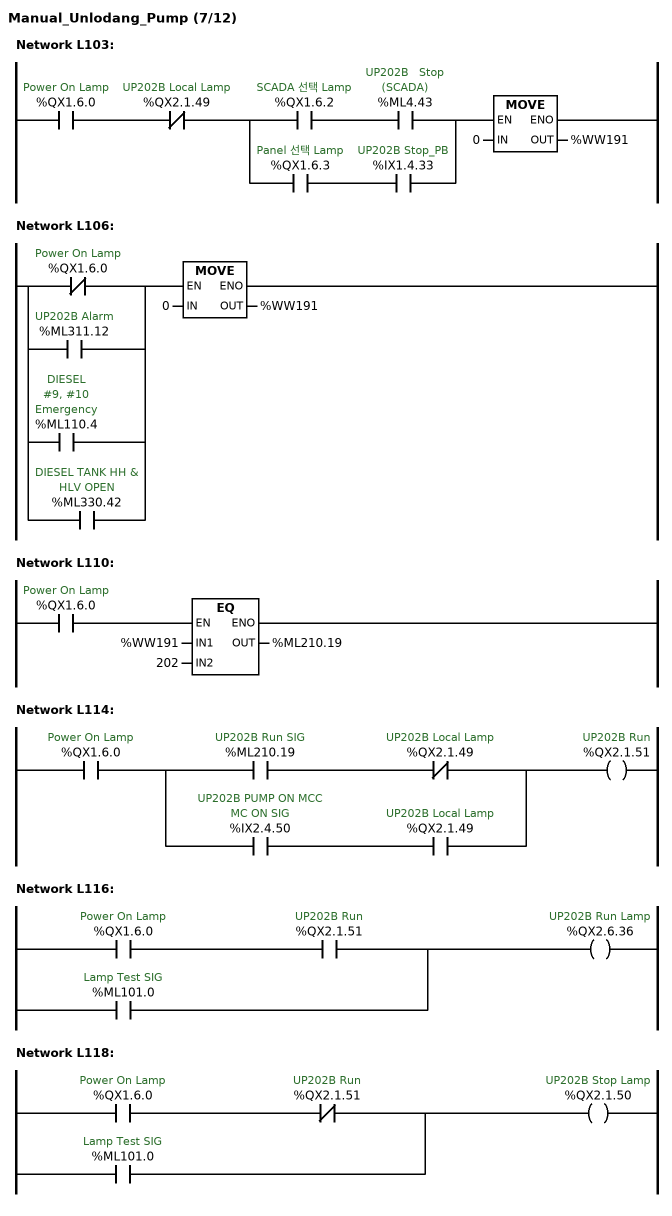
(* [picture p96: Manual_Unlodang_Pump rungs L103-L118] *)
(* Rung L103 *)
IF %QX1.6.0 AND NOT %QX2.1.49 AND ((%QX1.6.2 AND %ML4.43) OR (%QX1.6.3 AND %IX1.4.33)) THEN
    %WW191 := 0;
END_IF;
(* Rung L106 *)
IF NOT %QX1.6.0 OR %ML311.12 OR %ML110.4 OR %ML330.42 THEN %WW191 := 0; END_IF;
(* Rung L110 *)
IF %QX1.6.0 THEN %ML210.19 := %WW191 = 202; END_IF;
(* Rung L114 *)
%QX2.1.51 := %QX1.6.0 AND ((%ML210.19 AND NOT %QX2.1.49) OR (%IX2.4.50 AND %QX2.1.49));
(* Rung L116 *)
%QX2.6.36 := (%QX1.6.0 AND %QX2.1.51) OR %ML101.0;
(* Rung L118 *)
%QX2.1.50 := (%QX1.6.0 AND NOT %QX2.1.51) OR %ML101.0;

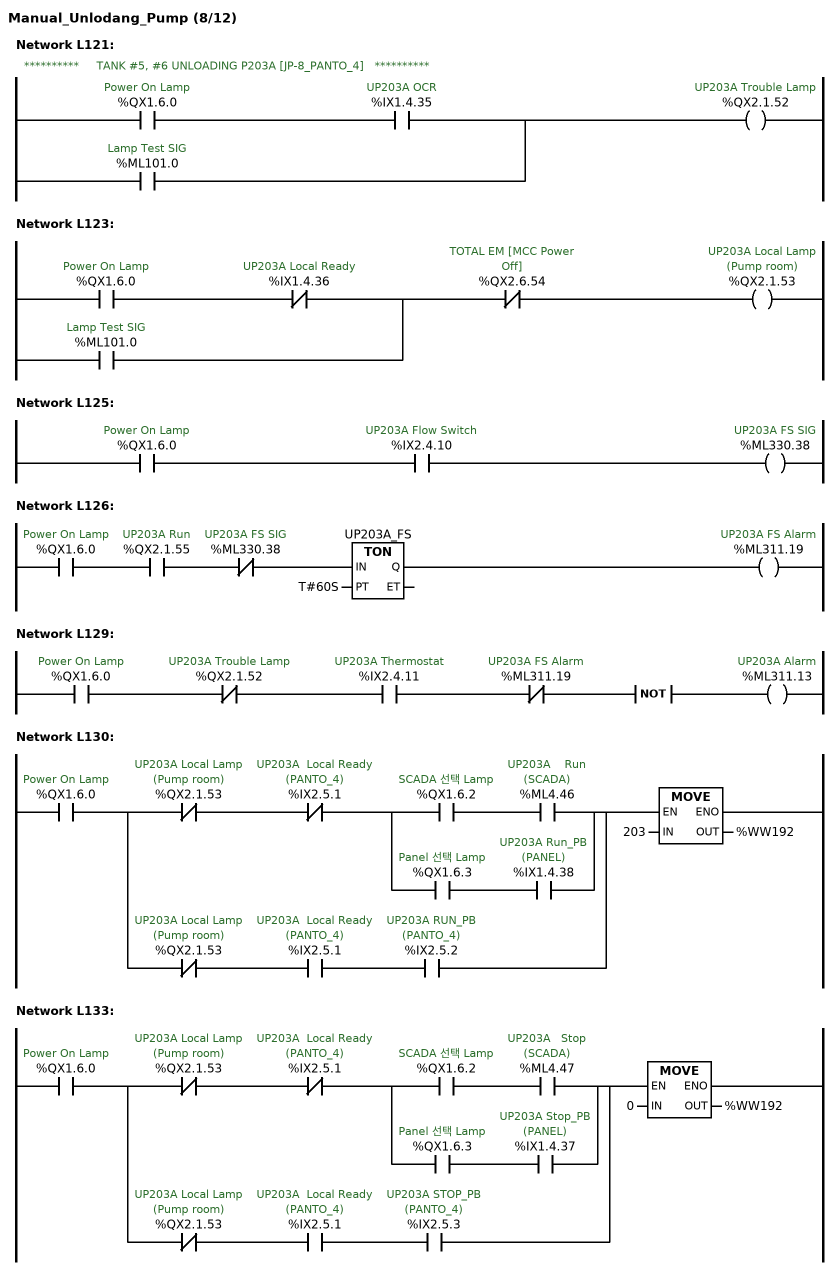
(* **********     TANK #5, #6 UNLOADING P203A [JP-8_PANTO_4]   ********** *)
(* Rung L121 *)
%QX2.1.52 := (%QX1.6.0 AND %IX1.4.35) OR %ML101.0;
(* Rung L123 *)
%QX2.1.53 := ((%QX1.6.0 AND NOT %IX1.4.36) OR %ML101.0) AND NOT %QX2.6.54;
(* Rung L125 *)
%ML330.38 := %QX1.6.0 AND %IX2.4.10;
(* Rung L126 *)
UP203A_FS(IN := %QX1.6.0 AND %QX2.1.55 AND NOT %ML330.38, PT := T#60S);
%ML311.19 := UP203A_FS.Q;
(* Rung L129 *)
%ML311.13 := NOT (%QX1.6.0 AND NOT %QX2.1.52 AND %IX2.4.11 AND NOT %ML311.19);
(* Rung L130 *)
IF %QX1.6.0 AND ((NOT %QX2.1.53 AND NOT %IX2.5.1 AND ((%QX1.6.2 AND %ML4.46) OR (%QX1.6.3 AND %IX1.4.38))) OR (NOT %QX2.1.53 AND %IX2.5.1 AND %IX2.5.2)) THEN
    %WW192 := 203;
END_IF;
(* Rung L133 *)
IF %QX1.6.0 AND ((NOT %QX2.1.53 AND NOT %IX2.5.1 AND ((%QX1.6.2 AND %ML4.47) OR (%QX1.6.3 AND %IX1.4.37))) OR (NOT %QX2.1.53 AND %IX2.5.1 AND %IX2.5.3)) THEN
    %WW192 := 0;
END_IF;

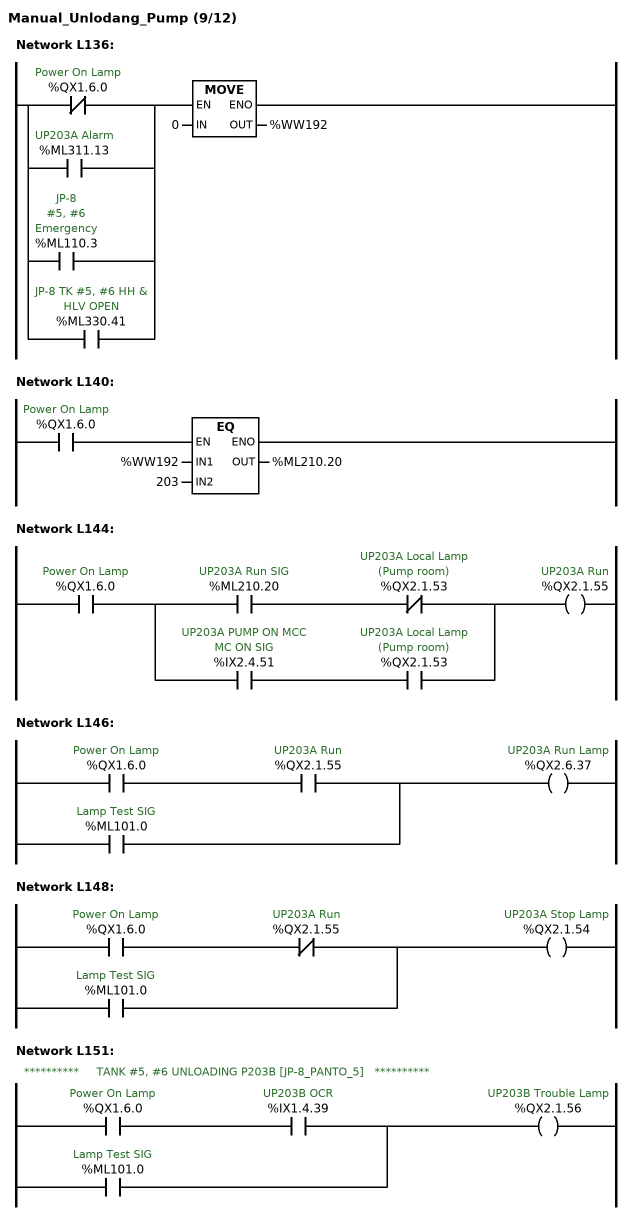
(* Rung L136 *)
IF NOT %QX1.6.0 OR %ML311.13 OR %ML110.3 OR %ML330.41 THEN %WW192 := 0; END_IF;
(* Rung L140 *)
IF %QX1.6.0 THEN %ML210.20 := %WW192 = 203; END_IF;
(* Rung L144 *)
%QX2.1.55 := %QX1.6.0 AND ((%ML210.20 AND NOT %QX2.1.53) OR (%IX2.4.51 AND %QX2.1.53));
(* Rung L146 *)
%QX2.6.37 := (%QX1.6.0 AND %QX2.1.55) OR %ML101.0;
(* Rung L148 *)
%QX2.1.54 := (%QX1.6.0 AND NOT %QX2.1.55) OR %ML101.0;
(* **********     TANK #5, #6 UNLOADING P203B [JP-8_PANTO_5]   ********** *)
(* Rung L151 *)
%QX2.1.56 := (%QX1.6.0 AND %IX1.4.39) OR %ML101.0;

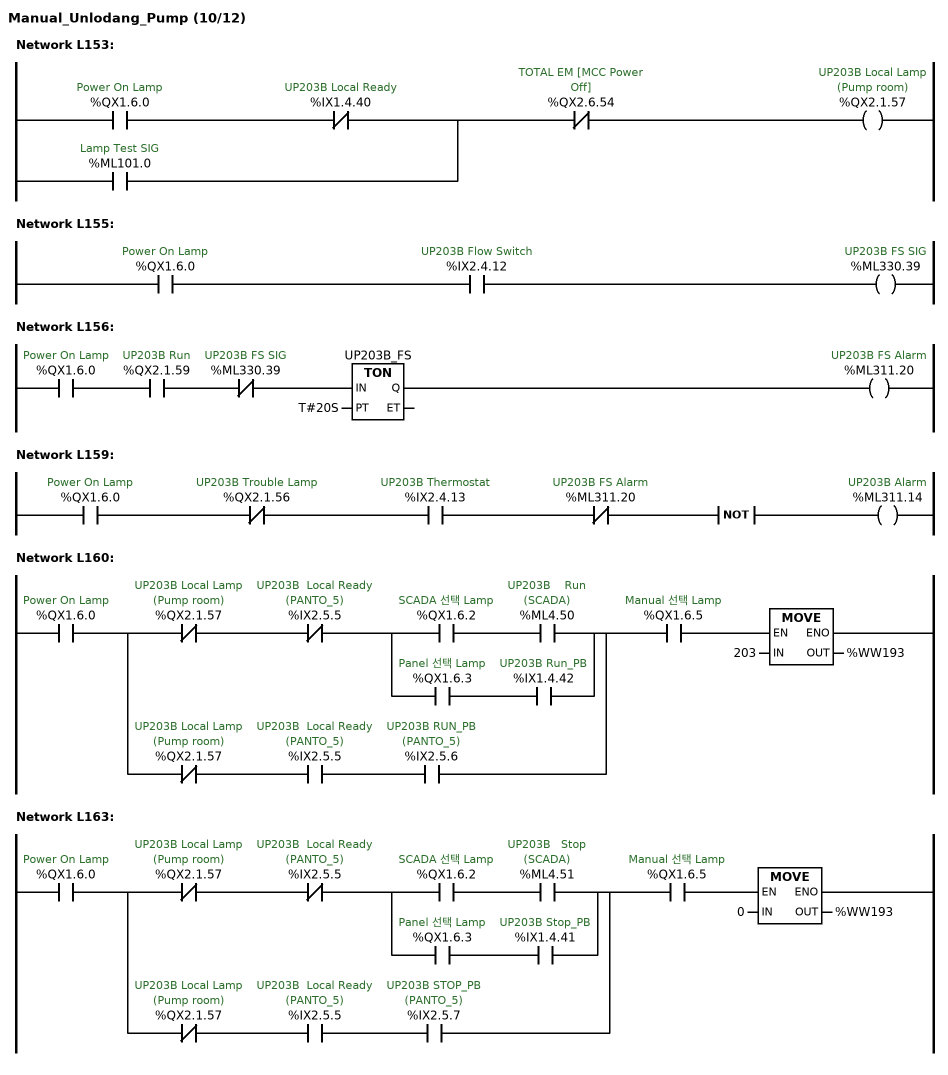
(* Rung L153 *)
%QX2.1.57 := ((%QX1.6.0 AND NOT %IX1.4.40) OR %ML101.0) AND NOT %QX2.6.54;
(* Rung L155 *)
%ML330.39 := %QX1.6.0 AND %IX2.4.12;
(* Rung L156 *)
UP203B_FS(IN := %QX1.6.0 AND %QX2.1.59 AND NOT %ML330.39, PT := T#20S);
%ML311.20 := UP203B_FS.Q;
(* Rung L159 *)
%ML311.14 := NOT (%QX1.6.0 AND NOT %QX2.1.56 AND %IX2.4.13 AND NOT %ML311.20);
(* Rung L160 *)
IF %QX1.6.0 AND ((NOT %QX2.1.57 AND NOT %IX2.5.5 AND ((%QX1.6.2 AND %ML4.50) OR (%QX1.6.3 AND %IX1.4.42))) OR (NOT %QX2.1.57 AND %IX2.5.5 AND %IX2.5.6)) AND %QX1.6.5 THEN
    %WW193 := 203;
END_IF;
(* Rung L163 *)
IF %QX1.6.0 AND ((NOT %QX2.1.57 AND NOT %IX2.5.5 AND ((%QX1.6.2 AND %ML4.51) OR (%QX1.6.3 AND %IX1.4.41))) OR (NOT %QX2.1.57 AND %IX2.5.5 AND %IX2.5.7)) AND %QX1.6.5 THEN
    %WW193 := 0;
END_IF;

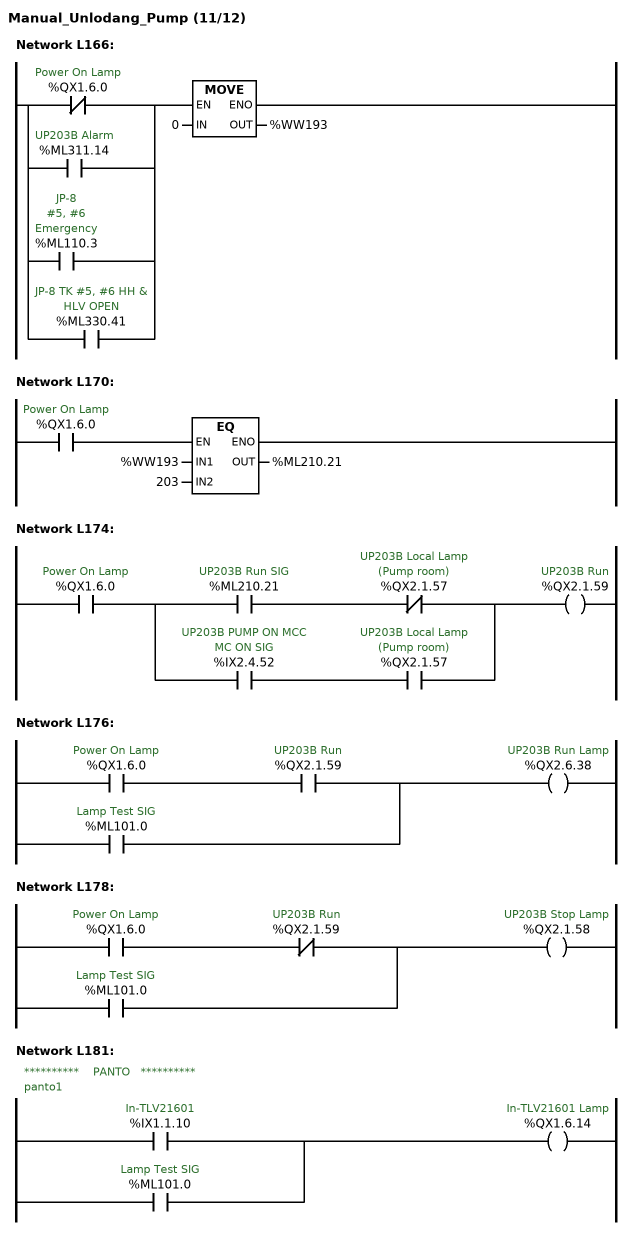
(* Rung L166 *)
IF NOT %QX1.6.0 OR %ML311.14 OR %ML110.3 OR %ML330.41 THEN %WW193 := 0; END_IF;
(* Rung L170 *)
IF %QX1.6.0 THEN %ML210.21 := %WW193 = 203; END_IF;
(* Rung L174 *)
%QX2.1.59 := %QX1.6.0 AND ((%ML210.21 AND NOT %QX2.1.57) OR (%IX2.4.52 AND %QX2.1.57));
(* Rung L176 *)
%QX2.6.38 := (%QX1.6.0 AND %QX2.1.59) OR %ML101.0;
(* Rung L178 *)
%QX2.1.58 := (%QX1.6.0 AND NOT %QX2.1.59) OR %ML101.0;
(* **********    PANTO   ********** *)
(* Rung L181 *)
%QX1.6.14 := %IX1.1.10 OR %ML101.0;
(* panto1 *)

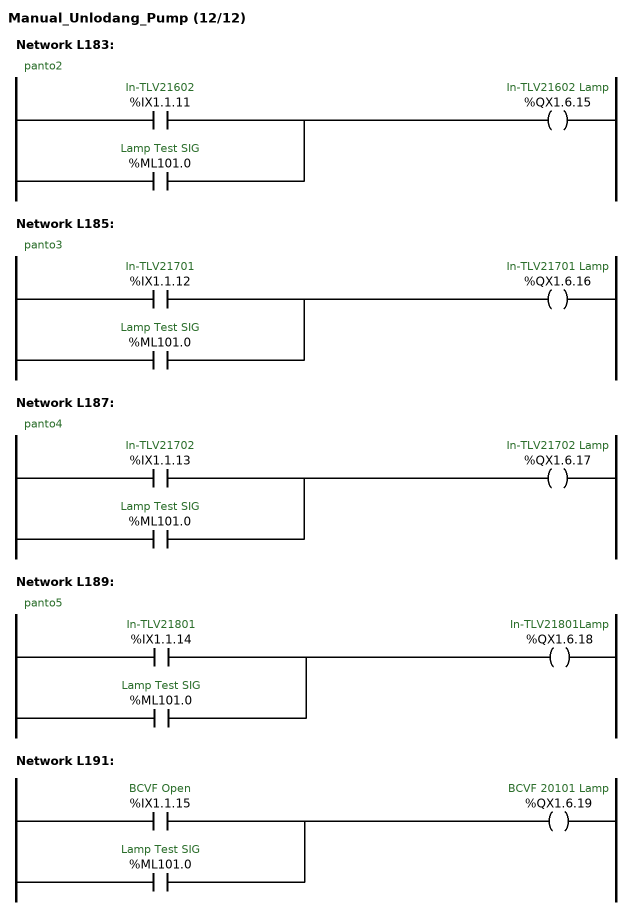
(* Rung L183 *)
%QX1.6.15 := %IX1.1.11 OR %ML101.0;
(* panto2 *)
(* Rung L185 *)
%QX1.6.16 := %IX1.1.12 OR %ML101.0;
(* panto3 *)
(* Rung L187 *)
%QX1.6.17 := %IX1.1.13 OR %ML101.0;
(* panto4 *)
(* Rung L189 *)
%QX1.6.18 := %IX1.1.14 OR %ML101.0;
(* panto5 *)
(* Rung L191 *)
%QX1.6.19 := %IX1.1.15 OR %ML101.0;
END_PROGRAM

PROGRAM ATG_LV_alarm_set (* task: 스캔 프로그램 *)
VAR
    tk001Water : WORD;
    tk002Water : WORD;
    tk003Water : WORD;
    tk101Water : WORD;
    tk102Water : WORD;
    tk103Water : WORD;
    tk104Water : WORD;
    tk105Water : WORD;
    tk106Water : WORD;
    tk107Water : WORD;
    tk108Water : WORD;
    tk109Water : WORD;
    tk110Water : WORD;
    tk111Water : WORD;
    tk112Water : WORD;
    tk113Water : WORD;
    tk401Water : WORD;
    tk402Water : WORD;
    tk403Water : WORD;
    tk404Water : WORD;
    TK_101_VOL : DWORD;
    TK_101_WAT : WORD;
    TK_102_VOL : DWORD;
    TK_103_VOL : DWORD;
    TK_104_VOL : DWORD;
    TK_105_VOL : DWORD;
    TK_106_VOL : DWORD;
    TK_107_VOL : DWORD;
    TK_108_VOL : DWORD;
    TK_109_VOL : DWORD;
    TK_110_VOL : DWORD;
    TK_401_VOL : DWORD;
    TK_402_VOL : DWORD;
    TK_403_VOL : DWORD;
    TK_404_VOL : DWORD;
END_VAR
VAR_EXTERNAL
    TK101H : DWORD;
    TK101HH : DWORD;
    TK101L : DWORD;
    TK101LL : DWORD;
    TK101VAL : DWORD;
    TK102H : DWORD;
    TK102HH : DWORD;
    TK102L : DWORD;
    TK102LL : DWORD;
    TK102VAL : DWORD;
    TK103H : DWORD;
    TK103HH : DWORD;
    TK103L : DWORD;
    TK103LL : DWORD;
    TK103VAL : DWORD;
    TK104H : DWORD;
    TK104HH : DWORD;
    TK104L : DWORD;
    TK104LL : DWORD;
    TK104VAL : DWORD;
    TK105H : DWORD;
    TK105HH : DWORD;
    TK105L : DWORD;
    TK105LL : DWORD;
    TK105VAL : DWORD;
    TK106H : DWORD;
    TK106HH : DWORD;
    TK106L : DWORD;
    TK106LL : DWORD;
    TK106VAL : DWORD;
    TK107H : DWORD;
    TK107HH : DWORD;
    TK107L : DWORD;
    TK107LL : DWORD;
    TK107VAL : DWORD;
    TK108H : DWORD;
    TK108HH : DWORD;
    TK108L : DWORD;
    TK108LL : DWORD;
    TK108VAL : DWORD;
    TK109H : DWORD;
    TK109HH : DWORD;
    TK109L : DWORD;
    TK109LL : DWORD;
    TK109VAL : DWORD;
    TK110H : DWORD;
    TK110HH : DWORD;
    TK110L : DWORD;
    TK110LL : DWORD;
    TK110VAL : DWORD;
    TK111H : DWORD;
    TK111HH : DWORD;
    TK111L : DWORD;
    TK111LL : DWORD;
    TK111VAL : DWORD;
    TK112H : DWORD;
    TK112HH : DWORD;
    TK112L : DWORD;
    TK112LL : DWORD;
    TK112VAL : DWORD;
    TK113H : DWORD;
    TK113HH : DWORD;
    TK113L : DWORD;
    TK113LL : DWORD;
    TK113VAL : DWORD;
END_VAR
// TANK 101 LEVEL ALARM SET //
TK101VAL:= %WD700 ; //REAL TIME TANK HEIGHT VALUE TO SCADA [DOUBLE WORD]
TK101HH := 7056 ; // HH LIMIT VALUE
TK101H  := 6371 ; // H LIMIT VALUE
TK101L  := 1583 ; // L LIMIT VALUE
TK101LL := 899  ; // LL LIMIT VALUE
%MX810(* 95% *) := TK101HH <  TK101VAL; // HOLDING [PRESS THE RESET BUTTON ON THE SCADA AND PANEL]
%MX811(* 90% *) := TK101HH >= TK101VAL AND TK101H  <= TK101VAL;
%MX813(* 15% *) := TK101L  >= TK101VAL AND TK101LL <= TK101VAL;
%MX814(* 10% *) := TK101LL >  TK101VAL; // HOLDING [PRESS THE RESET BUTTON ON THE SCADA AND PANEL]
%MX311 := %MX811; // REAL TIME HIGH ALARM
%MX313 := %MX813; // REAL TIME LOW

// TANK 102 LEVEL ALARM SET //
TK102VAL:= %WD710 ;
TK102HH := 7061 ; 
TK102H  := 6377 ; 
TK102L  := 1589 ; 
TK102LL := 905  ;
%MX820(* 95% *) := TK102HH <  TK102VAL ; // HOLDING [PRESS THE RESET BUTTON ON THE SCADA AND PANEL]
%MX821(* 90% *) := TK102HH >= TK102VAL AND TK102H  <= TK102VAL ;
%MX823(* 15% *) := TK102L  >= TK102VAL AND TK102LL <= TK102VAL ;
%MX824(* 10% *) := TK102LL >  TK102VAL ; // HOLDING [PRESS THE RESET BUTTON ON THE SCADA AND PANEL]
%MX321 := %MX821; // REAL TIME HIGH ALARM
%MX323 := %MX823; // REAL TIME LOW ALARM

// TANK 103 LEVEL ALARM SET //
TK103VAL:= %WD720 ;
TK103HH := 7063 ; 
TK103H  := 6378 ; 
TK103L  := 1589 ; 
TK103LL := 905  ;
%MX830(* 95% *) := TK103HH <  TK103VAL ; // HOLDING [PRESS THE RESET BUTTON ON THE SCADA AND PANEL]
%MX831(* 90% *) := TK103HH >= TK103VAL AND TK103H  <= TK103VAL ;
%MX833(* 15% *) := TK103L  >= TK103VAL AND TK103LL <= TK103VAL ;
%MX834(* 10% *) := TK103LL >  TK103VAL ; // HOLDING [PRESS THE RESET BUTTON ON THE SCADA AND PANEL]
%MX331 := %MX831; // REAL TIME HIGH ALARM
%MX333 := %MX833; // REAL TIME LOW ALARM

// TANK 104 LEVEL ALARM SET //
TK104VAL:= %WD730 ;
TK104HH := 7045 ; 
TK104H  := 6361 ; 
TK104L  := 1572 ; 
TK104LL := 888  ;
%MX840(* 95% *) := TK104HH <  TK104VAL ; // HOLDING [PRESS THE RESET BUTTON ON THE SCADA AND PANEL]
%MX841(* 90% *) := TK104HH >= TK104VAL AND TK104H  <= TK104VAL ;
%MX843(* 15% *) := TK104L  >= TK104VAL AND TK104LL <= TK104VAL ;
%MX844(* 10% *) := TK104LL >  TK104VAL ; // HOLDING [PRESS THE RESET BUTTON ON THE SCADA AND PANEL]
%MX341 := %MX841; // REAL TIME HIGH ALARM
%MX343 := %MX843; // REAL TIME LOW ALARM

// TANK 105 LEVEL ALARM SET //
TK105VAL:= %WD740 ;
TK105HH := 5256 ; 
TK105H  := 4713 ; 
TK105L  := 1186 ; 
TK105LL := 644  ;
%MX850(* 95% *) := TK105HH <  TK105VAL ; // HOLDING [PRESS THE RESET BUTTON ON THE SCADA AND PANEL]
%MX851(* 90% *) := TK105HH >= TK105VAL AND TK105H  <= TK105VAL ;
%MX853(* 15% *) := TK105L  >= TK105VAL AND TK105LL <= TK105VAL ;
%MX854(* 10% *) := TK105LL >  TK105VAL ; // HOLDING [PRESS THE RESET BUTTON ON THE SCADA AND PANEL]
%MX351 := %MX851; // REAL TIME HIGH ALARM
%MX353 := %MX853; // REAL TIME LOW ALARM

// TANK 106 LEVEL ALARM SET //
TK106VAL:= %WD750 ;
TK106HH := 5267 ; 
TK106H  := 4723 ; 
TK106L  := 1198 ; 
TK106LL := 656  ;
%MX860(* 95% *) := TK106HH <  TK106VAL ; // HOLDING [PRESS THE RESET BUTTON ON THE SCADA AND PANEL]
%MX861(* 90% *) := TK106HH >= TK106VAL AND TK106H  <= TK106VAL ;
%MX863(* 15% *) := TK106L  >= TK106VAL AND TK106LL <= TK106VAL ;
%MX864(* 10% *) := TK106LL >  TK106VAL ; // HOLDING [PRESS THE RESET BUTTON ON THE SCADA AND PANEL]
%MX361 := %MX861; // REAL TIME HIGH ALARM
%MX363 := %MX863; // REAL TIME LOW ALARM

// TANK 107 LEVEL ALARM SET //
TK107VAL:= %WD760 ;
TK107HH := 7177 ; 
TK107H  := 6493 ; 
TK107L  := 1697 ; 
TK107LL := 1012 ;
%MX870(* 95% *) := TK107HH <  TK107VAL ; // HOLDING [PRESS THE RESET BUTTON ON THE SCADA AND PANEL]
%MX871(* 90% *) := TK107HH >= TK107VAL AND TK107H  <= TK107VAL ;
%MX873(* 15% *) := TK107L  >= TK107VAL AND TK107LL <= TK107VAL ;
%MX874(* 10% *) := TK107LL >  TK107VAL ; // HOLDING [PRESS THE RESET BUTTON ON THE SCADA AND PANEL]
%MX371 := %MX871; // REAL TIME HIGH ALARM
%MX373 := %MX873; // REAL TIME LOW ALARM

// TANK 108 LEVEL ALARM SET //
TK108VAL:= %WD770 ;
TK108HH := 7172 ; 
TK108H  := 6487 ; 
TK108L  := 1693 ; 
TK108LL := 1008 ;
%MX880(* 95% *) := TK108HH <  TK108VAL ; // HOLDING [PRESS THE RESET BUTTON ON THE SCADA AND PANEL]
%MX881(* 90% *) := TK108HH >= TK108VAL AND TK108H  <= TK108VAL ;
%MX883(* 15% *) := TK108L  >= TK108VAL AND TK108LL <= TK108VAL ;
%MX884(* 10% *) := TK108LL >  TK108VAL ; // HOLDING [PRESS THE RESET BUTTON ON THE SCADA AND PANEL]
%MX381 := %MX881; // REAL TIME HIGH ALARM
%MX383 := %MX883; // REAL TIME LOW ALARM

// TANK 109 LEVEL ALARM SET //
TK109VAL:= %WD780 ;
TK109HH := 5144 ; 
TK109H  := 4609 ; 
TK109L  := 1127 ; 
TK109LL := 592  ;
%MX890(* 95% *) := TK109HH <  TK109VAL ; // HOLDING [PRESS THE RESET BUTTON ON THE SCADA AND PANEL]
%MX891(* 90% *) := TK109HH >= TK109VAL AND TK109H  <= TK109VAL ;
%MX893(* 15% *) := TK109L  >= TK109VAL AND TK109LL <= TK109VAL ;
%MX894(* 10% *) := TK109LL >  TK109VAL ; // HOLDING [PRESS THE RESET BUTTON ON THE SCADA AND PANEL]
%MX391 := %MX891; // REAL TIME HIGH ALARM
%MX393 := %MX893; // REAL TIME LOW ALARM

// TANK 110 LEVEL ALARM SET //
TK110VAL:= %WD790 ;
TK110HH := 5144 ; 
TK110H  := 4609 ; 
TK110L  := 1128 ; 
TK110LL := 592  ;
%MX900(* 95% *) := TK110HH <  TK110VAL ; // HOLDING [PRESS THE RESET BUTTON ON THE SCADA AND PANEL]
%MX901(* 90% *) := TK110HH >= TK110VAL AND TK110H  <= TK110VAL ;
%MX903(* 15% *) := TK110L  >= TK110VAL AND TK110LL <= TK110VAL ;
%MX904(* 10% *) := TK110LL >  TK110VAL ; // HOLDING [PRESS THE RESET BUTTON ON THE SCADA AND PANEL]
%MX401 := %MX901; // REAL TIME HIGH ALARM
%MX403 := %MX903; // REAL TIME LOW ALARM

// TANK 111 LEVEL ALARM SET //
%WD500  := WORD_TO_DWORD(IN:=%WW506);
TK111VAL:= %WD500 ;
TK111HH := 1578 ; 
TK111H  := 1398 ; 
TK111L  := 633 ; 
TK111LL := 440 ;
%MX910(* 95% *) := TK111HH <  TK111VAL ; // HOLDING [PRESS THE RESET BUTTON ON THE SCADA AND PANEL]
%MX911(* 90% *) := TK111HH >= TK111VAL AND TK111H  <= TK111VAL ;
%MX913(* 15% *) := TK111L  >= TK111VAL AND TK111LL <= TK111VAL ;
%MX914(* 10% *) := TK111LL >  TK111VAL ; // HOLDING [PRESS THE RESET BUTTON ON THE SCADA AND PANEL]
%MX411 := %MX911; // REAL TIME HIGH ALARM
%MX413 := %MX913; // REAL TIME LOW ALARM

// TANK 112 LEVEL ALARM SET //
%WD510  := WORD_TO_DWORD(IN:=%WW516);
TK112VAL:= %WD510 ;
TK112HH := 1100 ; //HLV 감지되는 실측 값 1175mm
TK112H  := 980; 
TK112L  := 491 ; 
TK112LL := 341 ;
%MX920(* 95% *) := TK112HH <  TK112VAL ; // HOLDING [PRESS THE RESET BUTTON ON THE SCADA AND PANEL]
%MX921(* 90% *) := TK112HH >= TK112VAL AND TK112H  <= TK112VAL ;
%MX923(* 15% *) := TK112L  >= TK112VAL AND TK112LL <= TK112VAL ;
%MX924(* 10% *) := TK112LL >  TK112VAL ; // HOLDING [PRESS THE RESET BUTTON ON THE SCADA AND PANEL]
%MX421 := %MX921; // REAL TIME HIGH ALARM
%MX423 := %MX923; // REAL TIME LOW ALARM

// TANK 113 LEVEL ALARM SET //
%WD520  := WORD_TO_DWORD(IN:=%WW526);
TK113VAL:= %WD520 ;
TK113HH := 1030 ; //HLV 감지되는 실측 값 1163mm
TK113H  := 904 ; 
TK113L  := 465 ; 
TK113LL := 323 ;
%MX930(* 95% *) := TK113HH <  TK113VAL ; // HOLDING [PRESS THE RESET BUTTON ON THE SCADA AND PANEL]
%MX931(* 90% *) := TK113HH >= TK113VAL AND TK113H  <= TK113VAL ;
%MX933(* 15% *) := TK113L  >= TK113VAL AND TK113LL <= TK113VAL ;
%MX934(* 10% *) := TK113LL >  TK113VAL ; // HOLDING [PRESS THE RESET BUTTON ON THE SCADA AND PANEL]
%MX431 := %MX931; // REAL TIME HIGH ALARM
%MX433 := %MX933; // REAL TIME LOW ALARM

// TANK VOLUME (PLC TO SCADA) //
TK_101_VOL := WORD_DWORD(LOW:=%WW603,HIGH:=%WW602); //TK-101 [%WD708 TO SCADA]
TK_102_VOL := WORD_DWORD(LOW:=%WW607,HIGH:=%WW606); //TK-102 [%WD718 TO SCADA]
TK_103_VOL := WORD_DWORD(LOW:=%WW611,HIGH:=%WW610); //TK-103 [%WD728 TO SCADA]
TK_104_VOL := WORD_DWORD(LOW:=%WW615,HIGH:=%WW614); //TK-104 [%WD738 TO SCADA]
TK_105_VOL := WORD_DWORD(LOW:=%WW619,HIGH:=%WW618); //TK-105 [%WD748 TO SCADA]
TK_106_VOL := WORD_DWORD(LOW:=%WW623,HIGH:=%WW622); //TK-106 [%WD758 TO SCADA]
TK_107_VOL := WORD_DWORD(LOW:=%WW627,HIGH:=%WW626); //TK-107 [%WD768 TO SCADA]
TK_108_VOL := WORD_DWORD(LOW:=%WW631,HIGH:=%WW630); //TK-108 [%WD778 TO SCADA]
TK_109_VOL := WORD_DWORD(LOW:=%WW635,HIGH:=%WW634); //TK-109 [%WD788 TO SCADA]
TK_110_VOL := WORD_DWORD(LOW:=%WW639,HIGH:=%WW638); //TK-110 [%WD798 TO SCADA]
%WW1100 := %WW506; //TK-111
%WW1103 := %WW516; //TK-112
%WW1106 := %WW526; //TK-113
TK_401_VOL := WORD_DWORD(LOW:=%WW655,HIGH:=%WW654); //TK-401 (120대대)  [%WD654 TO SCADA]
TK_402_VOL := WORD_DWORD(LOW:=%WW659,HIGH:=%WW658); //TK-402 (121대대)  [%WD658 TO SCADA]
TK_403_VOL := WORD_DWORD(LOW:=%WW663,HIGH:=%WW662); //TK-403 (123대대)  [%WD662 TO SCADA]
TK_404_VOL := WORD_DWORD(LOW:=%WW667,HIGH:=%WW666); //TK-404 (157대대)  [%WD666 TO SCADA]

// PLC TO SCADA (DWORD) //
%WD708 := TK_101_VOL;
%WD718 := TK_102_VOL;
%WD728 := TK_103_VOL;
%WD738 := TK_104_VOL;
%WD748 := TK_105_VOL;
%WD758 := TK_106_VOL;
%WD768 := TK_107_VOL;
%WD778 := TK_108_VOL;
%WD788 := TK_109_VOL;
%WD798 := TK_110_VOL;

%WD654 := TK_401_VOL;
%WD658 := TK_402_VOL;
%WD662 := TK_403_VOL;
%WD666 := TK_404_VOL;

// PLC TO SCADA (WATER LEVEL) //
// POL TANK ARES
tk101Water := %WW601;
tk102Water := %WW605;
tk103Water := %WW609;
tk104Water := %WW613;
tk107Water := %WW625;
tk108Water := %WW629;
// POL JP-8
tk105Water := %WW617;
tk106Water := %WW621;
// POL DIESEL
tk109Water := %WW633;
tk110Water := %WW637;
// POL DRAIN
tk111Water := %WW641; //ARES
tk112Water := %WW645; //JP-8
tk113Water := %WW649; //DIESEL
// SQUAD
tk401Water := %WW653; //SQ 120
tk402Water := %WW657; //SQ 121
tk403Water := %WW661; //SQ 123
tk404Water := %WW665; //SQ 157
//HONG SUNG
tk001Water := %WW669; //BUFFER
tk002Water := %WW673; //MAIN
tk003Water := %WW677; //DRAIN
END_PROGRAM

PROGRAM Analog (* task: 스캔 프로그램 *)
VAR_EXTERNAL
    _0100_CH0_ACT : BOOL; (* AT %UX1.0.16 *) (* 아날로그입력 모듈: 채널0 운전중 *)
    _0100_CH0_DATA : INT; (* AT %UW1.0.2 *) (* 아날로그입력 모듈: 채널0 변환값 *)
    _0100_CH0_IDD : BOOL; (* AT %UX1.0.160 *) (* 아날로그입력 모듈: 채널0 입력단선검출 *)
    _0100_CH1_ACT : BOOL; (* AT %UX1.0.17 *) (* 아날로그입력 모듈: 채널1 운전중 *)
    _0100_CH1_DATA : INT; (* AT %UW1.0.3 *) (* 아날로그입력 모듈: 채널1 변환값 *)
    _0100_CH1_IDD : BOOL; (* AT %UX1.0.161 *) (* 아날로그입력 모듈: 채널1 입력단선검출 *)
    _0100_CH2_ACT : BOOL; (* AT %UX1.0.18 *) (* 아날로그입력 모듈: 채널2 운전중 *)
    _0100_CH2_DATA : INT; (* AT %UW1.0.4 *) (* 아날로그입력 모듈: 채널2 변환값 *)
    _0100_CH2_IDD : BOOL; (* AT %UX1.0.162 *) (* 아날로그입력 모듈: 채널2 입력단선검출 *)
    _0100_CH3_ACT : BOOL; (* AT %UX1.0.19 *) (* 아날로그입력 모듈: 채널3 운전중 *)
    _0100_CH3_DATA : INT; (* AT %UW1.0.5 *) (* 아날로그입력 모듈: 채널3 변환값 *)
    _0100_CH3_IDD : BOOL; (* AT %UX1.0.163 *) (* 아날로그입력 모듈: 채널3 입력단선검출 *)
    _0100_CH4_ACT : BOOL; (* AT %UX1.0.20 *) (* 아날로그입력 모듈: 채널4 운전중 *)
    _0100_CH4_DATA : INT; (* AT %UW1.0.6 *) (* 아날로그입력 모듈: 채널4 변환값 *)
    _0100_CH4_IDD : BOOL; (* AT %UX1.0.164 *) (* 아날로그입력 모듈: 채널4 입력단선검출 *)
    _0100_CH5_ACT : BOOL; (* AT %UX1.0.21 *) (* 아날로그입력 모듈: 채널5 운전중 *)
    _0100_CH5_DATA : INT; (* AT %UW1.0.7 *) (* 아날로그입력 모듈: 채널5 변환값 *)
    _0100_CH5_IDD : BOOL; (* AT %UX1.0.165 *) (* 아날로그입력 모듈: 채널5 입력단선검출 *)
    _0100_CH6_ACT : BOOL; (* AT %UX1.0.22 *) (* 아날로그입력 모듈: 채널6 운전중 *)
    _0100_CH6_DATA : INT; (* AT %UW1.0.8 *) (* 아날로그입력 모듈: 채널6 변환값 *)
    _0100_CH6_IDD : BOOL; (* AT %UX1.0.166 *) (* 아날로그입력 모듈: 채널6 입력단선검출 *)
    _0100_CH7_ACT : BOOL; (* AT %UX1.0.23 *) (* 아날로그입력 모듈: 채널7 운전중 *)
    _0100_CH7_DATA : INT; (* AT %UW1.0.9 *) (* 아날로그입력 모듈: 채널7 변환값 *)
    _0100_CH7_IDD : BOOL; (* AT %UX1.0.167 *) (* 아날로그입력 모듈: 채널7 입력단선검출 *)
    _0208_CH0_ACT : BOOL; (* AT %UX2.8.16 *) (* 아날로그출력 모듈: 채널0 운전중 *)
    _0208_CH0_DATA : INT; (* AT %UW2.8.3 *) (* 아날로그출력 모듈: 채널0 입력값 *)
    _0208_CH0_ERR : BOOL; (* AT %UX2.8.0 *) (* 아날로그출력 모듈: 채널0 에러 *)
    _0208_CH0_OUTEN : BOOL; (* AT %UX2.8.32 *) (* 아날로그출력 모듈: 채널0 출력상태설정 *)
END_VAR
VAR
    _PT102_ADJ : DWORD;
END_VAR
VAR
    _t1 : BOOL;
    _t2 : BOOL;
    _t3 : BOOL;
    _t4 : BOOL;
END_VAR

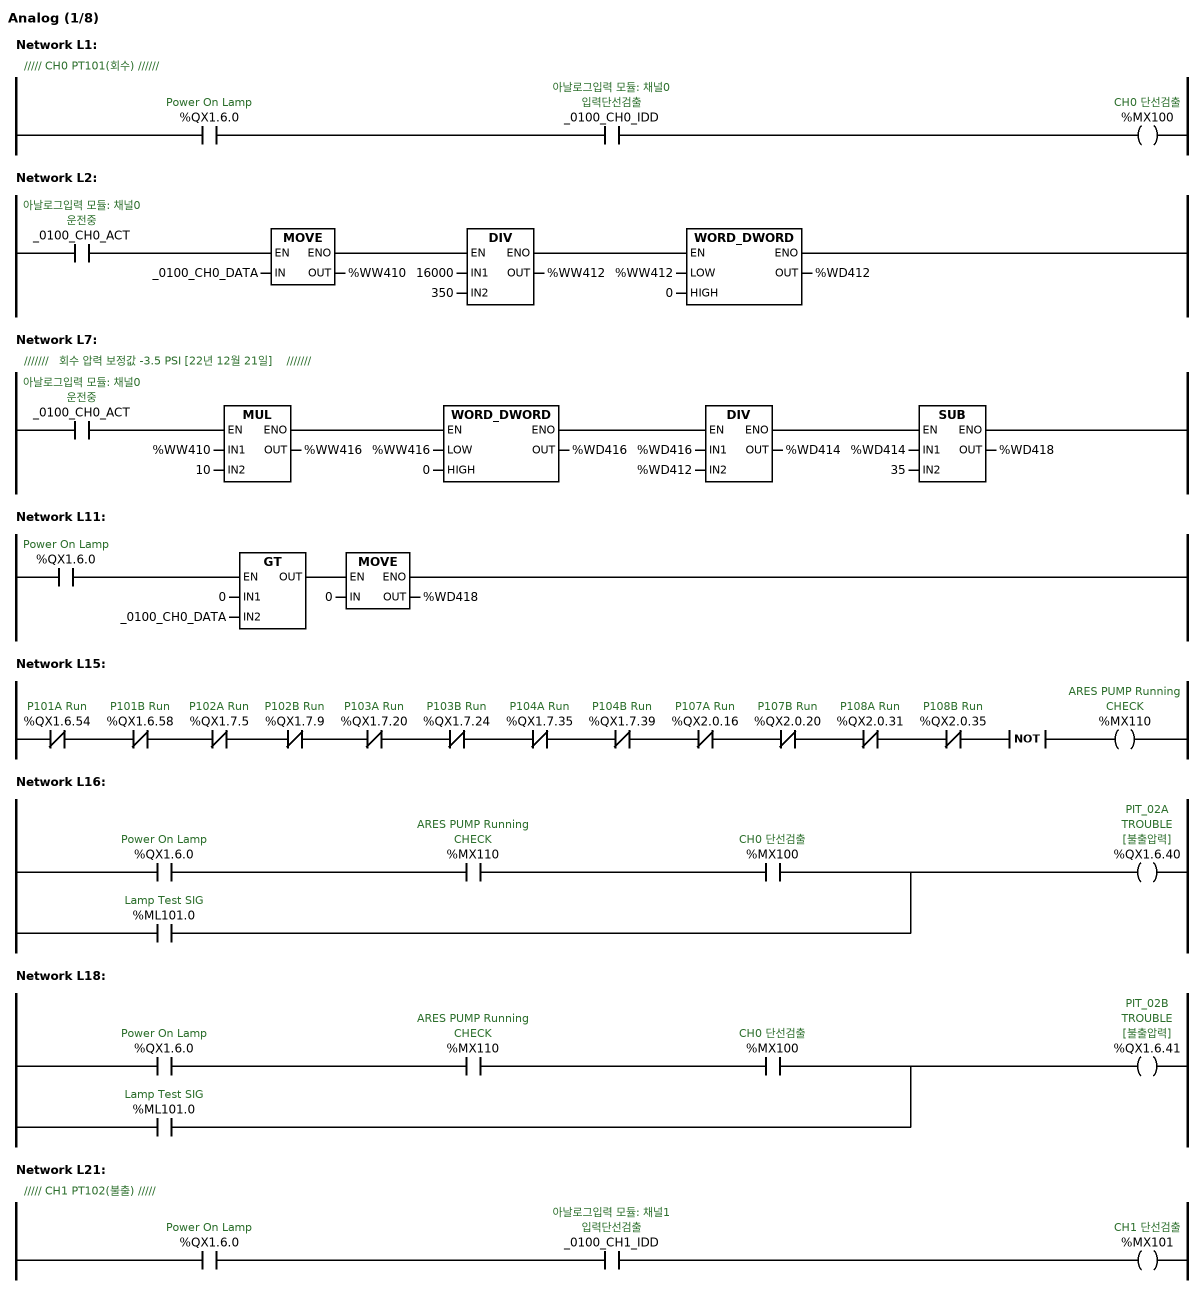
(* ///// CH0 PT101(회수) ////// *)
(* Rung L1 *)
%MX100 := %QX1.6.0 AND _0100_CH0_IDD;
(* Rung L2 *)
IF _0100_CH0_ACT THEN
    %WW410 := _0100_CH0_DATA;
    %WW412 := 16000 / 350;
    %WD412 := WORD_DWORD(LOW := %WW412, HIGH := 0);
END_IF;
(* ///////   회수 압력 보정값 -3.5 PSI [22년 12월 21일]    /////// *)
(* Rung L7 *)
IF _0100_CH0_ACT THEN
    %WW416 := %WW410 * 10;
    %WD416 := WORD_DWORD(LOW := %WW416, HIGH := 0);
    %WD414 := %WD416 / %WD412;
    %WD418 := %WD414 - 35;
END_IF;
(* Rung L11 *)
IF %QX1.6.0 THEN _t1 := 0 > _0100_CH0_DATA; END_IF;
IF _t1 THEN %WD418 := 0; END_IF;
(* Rung L15 *)
%MX110 := NOT (NOT %QX1.6.54 AND NOT %QX1.6.58 AND NOT %QX1.7.5 AND NOT %QX1.7.9 AND NOT %QX1.7.20 AND NOT %QX1.7.24 AND NOT %QX1.7.35 AND NOT %QX1.7.39 AND NOT %QX2.0.16 AND NOT %QX2.0.20 AND NOT %QX2.0.31 AND NOT %QX2.0.35);
(* Rung L16 *)
%QX1.6.40 := (%QX1.6.0 AND %MX110 AND %MX100) OR %ML101.0;
(* Rung L18 *)
%QX1.6.41 := (%QX1.6.0 AND %MX110 AND %MX100) OR %ML101.0;
(* ///// CH1 PT102(불출) ///// *)
(* Rung L21 *)
%MX101 := %QX1.6.0 AND _0100_CH1_IDD;

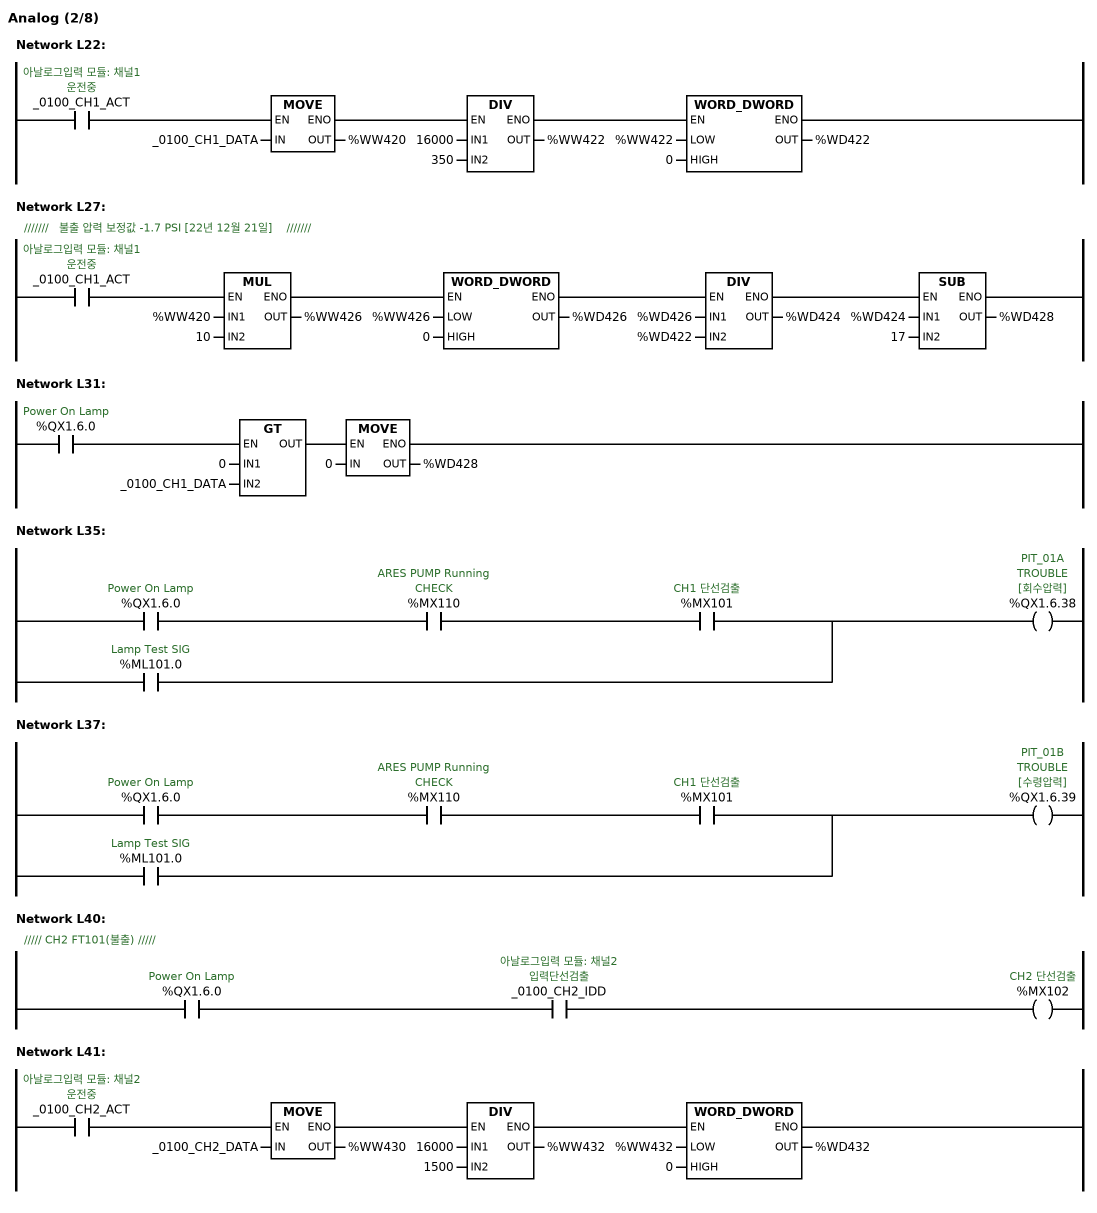
(* Rung L22 *)
IF _0100_CH1_ACT THEN
    %WW420 := _0100_CH1_DATA;
    %WW422 := 16000 / 350;
    %WD422 := WORD_DWORD(LOW := %WW422, HIGH := 0);
END_IF;
(* ///////   불출 압력 보정값 -1.7 PSI [22년 12월 21일]    /////// *)
(* Rung L27 *)
IF _0100_CH1_ACT THEN
    %WW426 := %WW420 * 10;
    %WD426 := WORD_DWORD(LOW := %WW426, HIGH := 0);
    %WD424 := %WD426 / %WD422;
    %WD428 := %WD424 - 17;
END_IF;
(* Rung L31 *)
IF %QX1.6.0 THEN _t2 := 0 > _0100_CH1_DATA; END_IF;
IF _t2 THEN %WD428 := 0; END_IF;
(* Rung L35 *)
%QX1.6.38 := (%QX1.6.0 AND %MX110 AND %MX101) OR %ML101.0;
(* Rung L37 *)
%QX1.6.39 := (%QX1.6.0 AND %MX110 AND %MX101) OR %ML101.0;
(* ///// CH2 FT101(불출) ///// *)
(* Rung L40 *)
%MX102 := %QX1.6.0 AND _0100_CH2_IDD;
(* Rung L41 *)
IF _0100_CH2_ACT THEN
    %WW430 := _0100_CH2_DATA;
    %WW432 := 16000 / 1500;
    %WD432 := WORD_DWORD(LOW := %WW432, HIGH := 0);
END_IF;

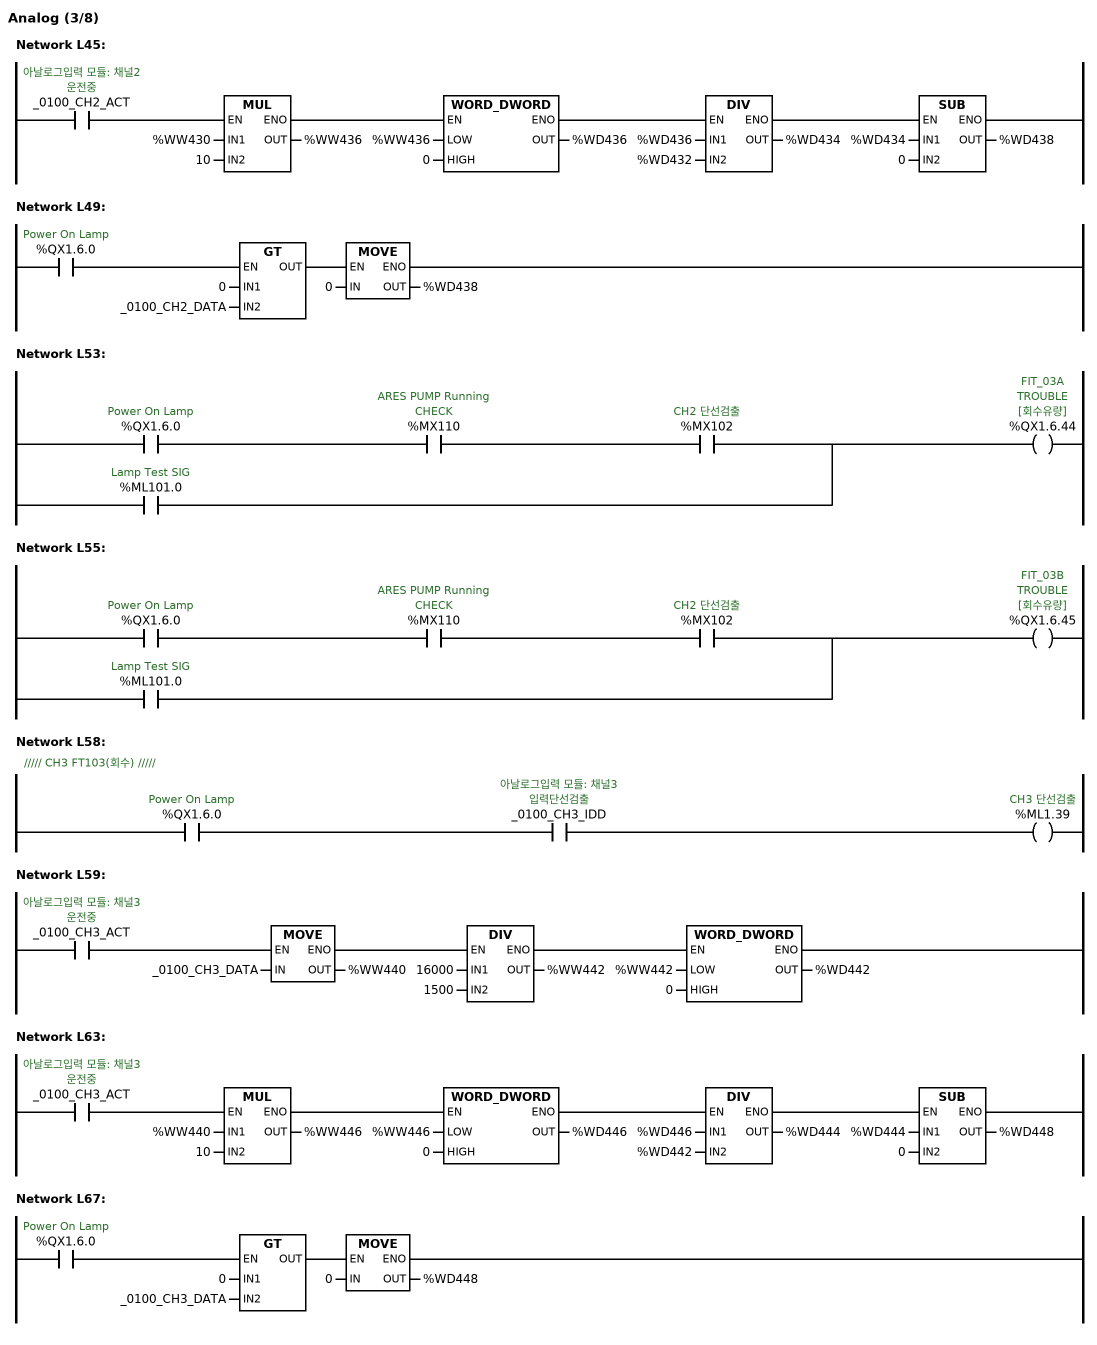
(* Rung L45 *)
IF _0100_CH2_ACT THEN
    %WW436 := %WW430 * 10;
    %WD436 := WORD_DWORD(LOW := %WW436, HIGH := 0);
    %WD434 := %WD436 / %WD432;
    %WD438 := %WD434 - 0;
END_IF;
(* Rung L49 *)
IF %QX1.6.0 THEN _t3 := 0 > _0100_CH2_DATA; END_IF;
IF _t3 THEN %WD438 := 0; END_IF;
(* Rung L53 *)
%QX1.6.44 := (%QX1.6.0 AND %MX110 AND %MX102) OR %ML101.0;
(* Rung L55 *)
%QX1.6.45 := (%QX1.6.0 AND %MX110 AND %MX102) OR %ML101.0;
(* ///// CH3 FT103(회수) ///// *)
(* Rung L58 *)
%ML1.39 := %QX1.6.0 AND _0100_CH3_IDD;
(* Rung L59 *)
IF _0100_CH3_ACT THEN
    %WW440 := _0100_CH3_DATA;
    %WW442 := 16000 / 1500;
    %WD442 := WORD_DWORD(LOW := %WW442, HIGH := 0);
END_IF;
(* Rung L63 *)
IF _0100_CH3_ACT THEN
    %WW446 := %WW440 * 10;
    %WD446 := WORD_DWORD(LOW := %WW446, HIGH := 0);
    %WD444 := %WD446 / %WD442;
    %WD448 := %WD444 - 0;
END_IF;
(* Rung L67 *)
IF %QX1.6.0 THEN _t4 := 0 > _0100_CH3_DATA; END_IF;
IF _t4 THEN %WD448 := 0; END_IF;

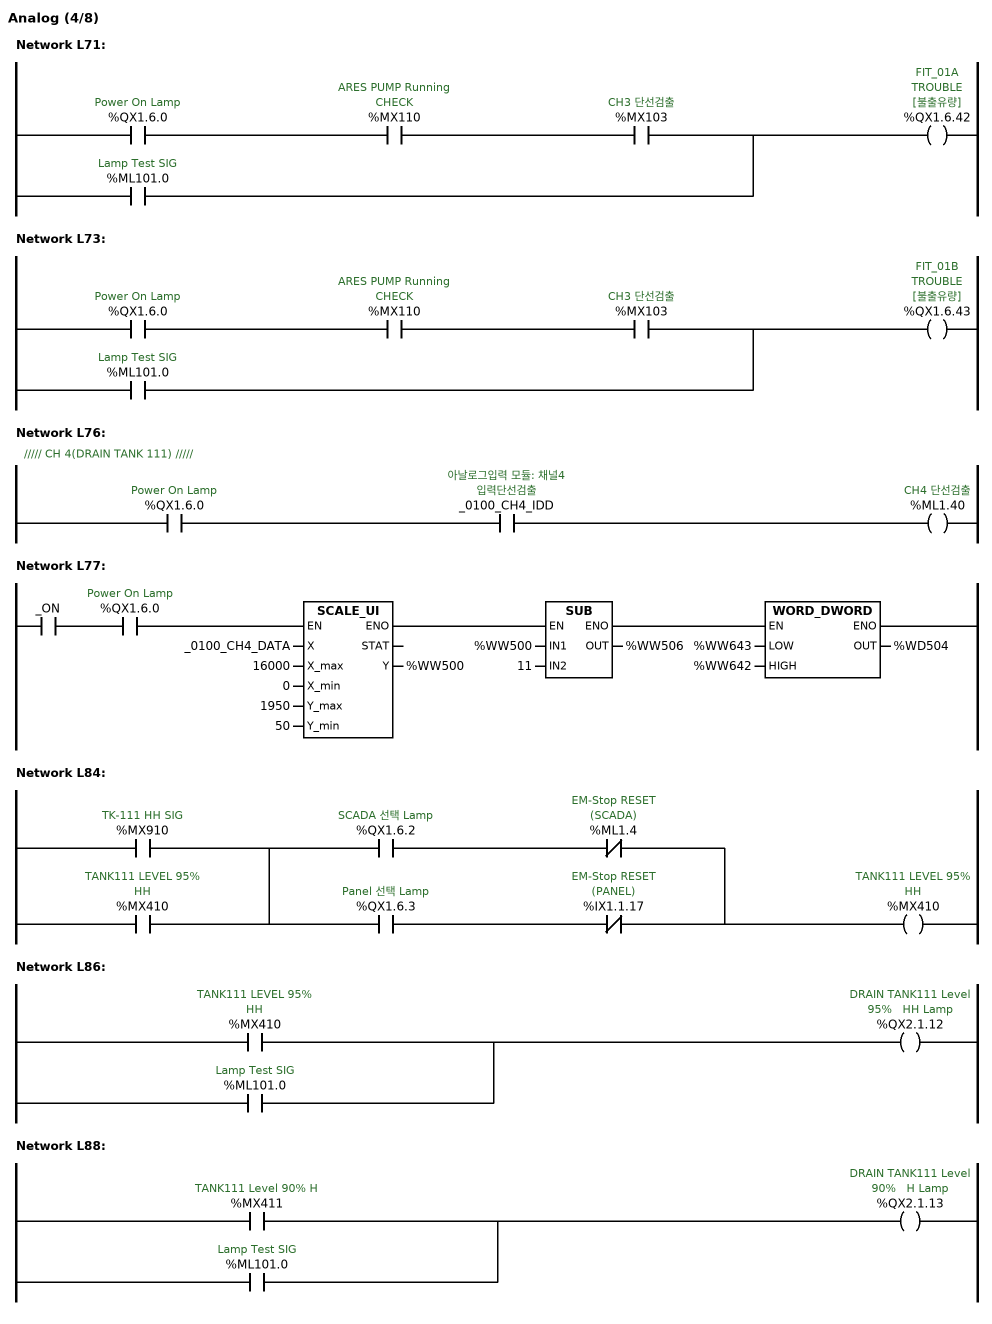
(* Rung L71 *)
%QX1.6.42 := (%QX1.6.0 AND %MX110 AND %MX103) OR %ML101.0;
(* Rung L73 *)
%QX1.6.43 := (%QX1.6.0 AND %MX110 AND %MX103) OR %ML101.0;
(* ///// CH 4(DRAIN TANK 111) ///// *)
(* Rung L76 *)
%ML1.40 := %QX1.6.0 AND _0100_CH4_IDD;
(* Rung L77 *)
IF _ON AND %QX1.6.0 THEN
    SCALE_UI(X := _0100_CH4_DATA, X_max := 16000, X_min := 0, Y_max := 1950, Y_min := 50, Y => %WW500);
    %WW506 := %WW500 - 11;
    %WD504 := WORD_DWORD(LOW := %WW643, HIGH := %WW642);
END_IF;
(* Rung L84 *)
%MX410 := (%MX910 OR %MX410) AND ((%QX1.6.2 AND NOT %ML1.4) OR (%QX1.6.3 AND NOT %IX1.1.17));
(* Rung L86 *)
%QX2.1.12 := %MX410 OR %ML101.0;
(* Rung L88 *)
%QX2.1.13 := %MX411 OR %ML101.0;

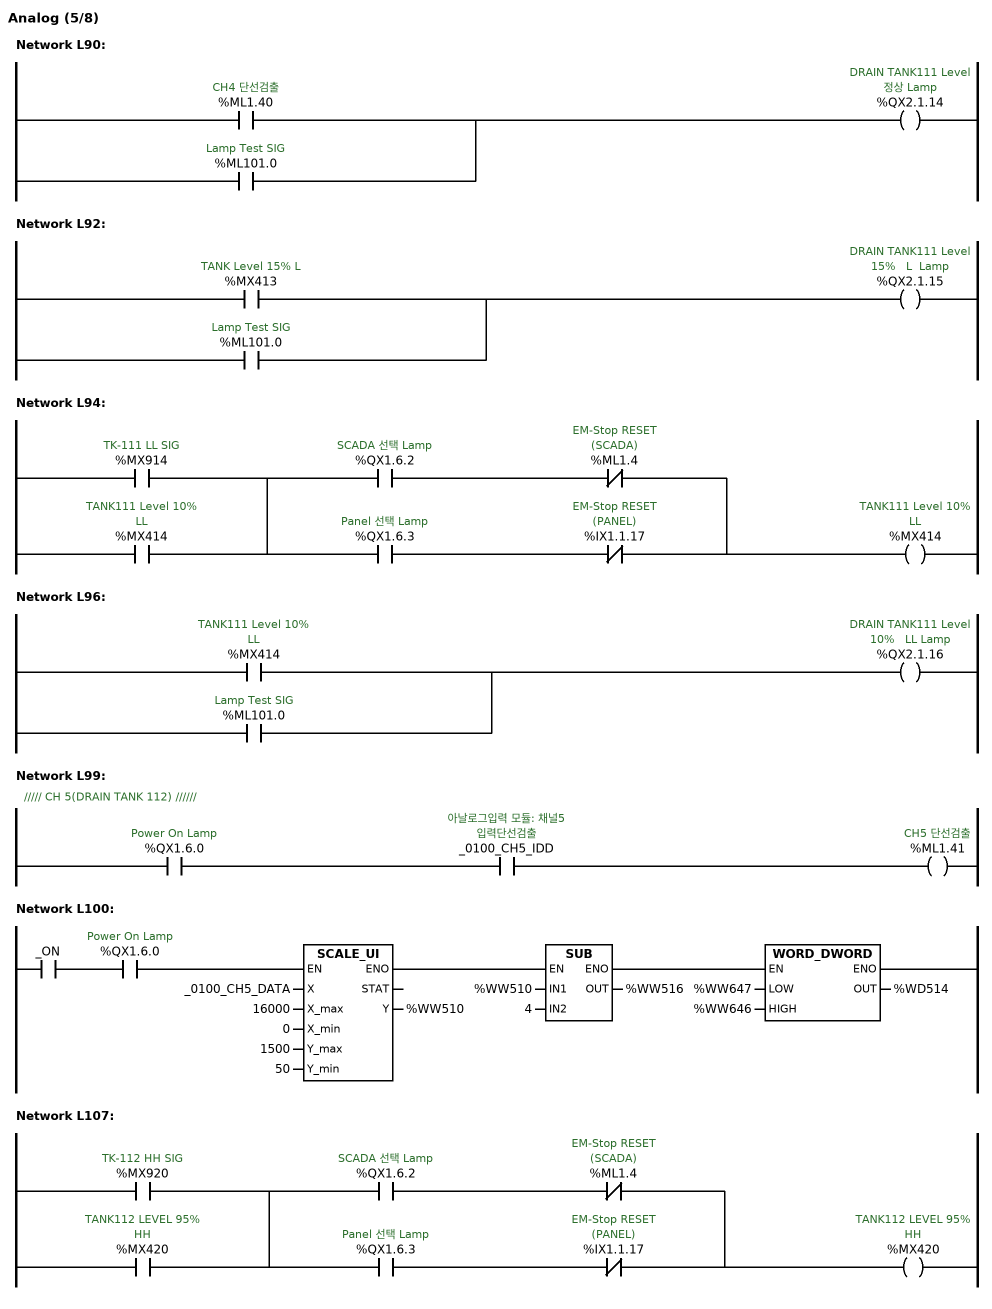
(* Rung L90 *)
%QX2.1.14 := %ML1.40 OR %ML101.0;
(* Rung L92 *)
%QX2.1.15 := %MX413 OR %ML101.0;
(* Rung L94 *)
%MX414 := (%MX914 OR %MX414) AND ((%QX1.6.2 AND NOT %ML1.4) OR (%QX1.6.3 AND NOT %IX1.1.17));
(* Rung L96 *)
%QX2.1.16 := %MX414 OR %ML101.0;
(* ///// CH 5(DRAIN TANK 112) ////// *)
(* Rung L99 *)
%ML1.41 := %QX1.6.0 AND _0100_CH5_IDD;
(* Rung L100 *)
IF _ON AND %QX1.6.0 THEN
    SCALE_UI(X := _0100_CH5_DATA, X_max := 16000, X_min := 0, Y_max := 1500, Y_min := 50, Y => %WW510);
    %WW516 := %WW510 - 4;
    %WD514 := WORD_DWORD(LOW := %WW647, HIGH := %WW646);
END_IF;
(* Rung L107 *)
%MX420 := (%MX920 OR %MX420) AND ((%QX1.6.2 AND NOT %ML1.4) OR (%QX1.6.3 AND NOT %IX1.1.17));

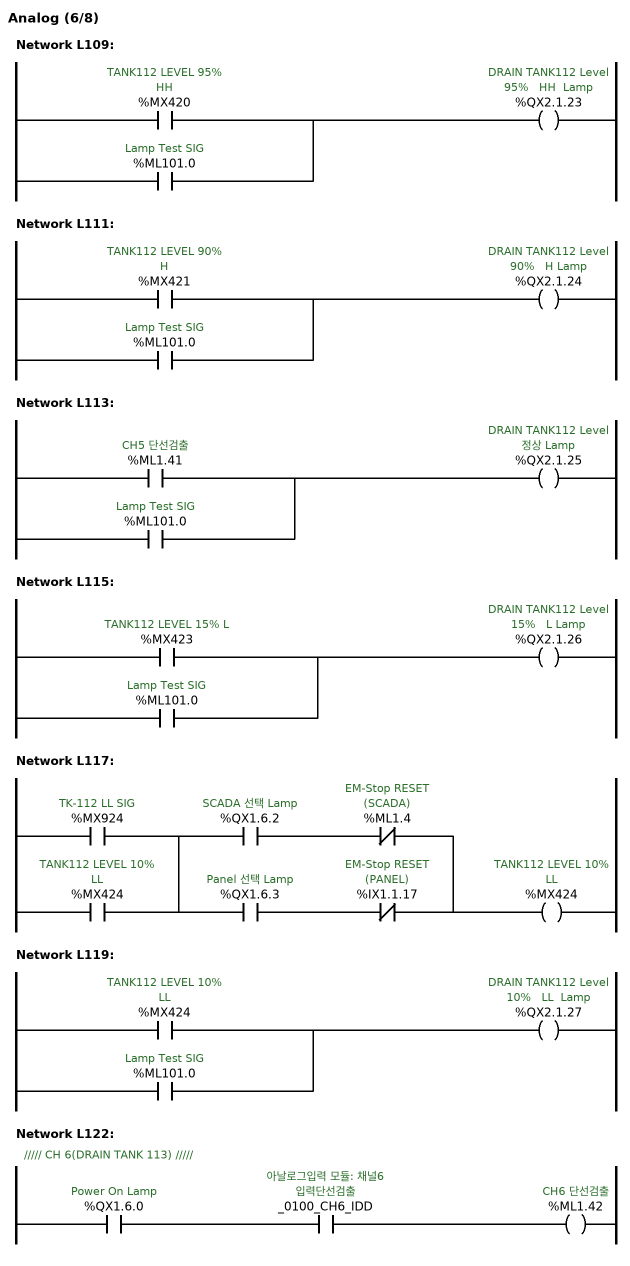
(* Rung L109 *)
%QX2.1.23 := %MX420 OR %ML101.0;
(* Rung L111 *)
%QX2.1.24 := %MX421 OR %ML101.0;
(* Rung L113 *)
%QX2.1.25 := %ML1.41 OR %ML101.0;
(* Rung L115 *)
%QX2.1.26 := %MX423 OR %ML101.0;
(* Rung L117 *)
%MX424 := (%MX924 OR %MX424) AND ((%QX1.6.2 AND NOT %ML1.4) OR (%QX1.6.3 AND NOT %IX1.1.17));
(* Rung L119 *)
%QX2.1.27 := %MX424 OR %ML101.0;
(* ///// CH 6(DRAIN TANK 113) ///// *)
(* Rung L122 *)
%ML1.42 := %QX1.6.0 AND _0100_CH6_IDD;

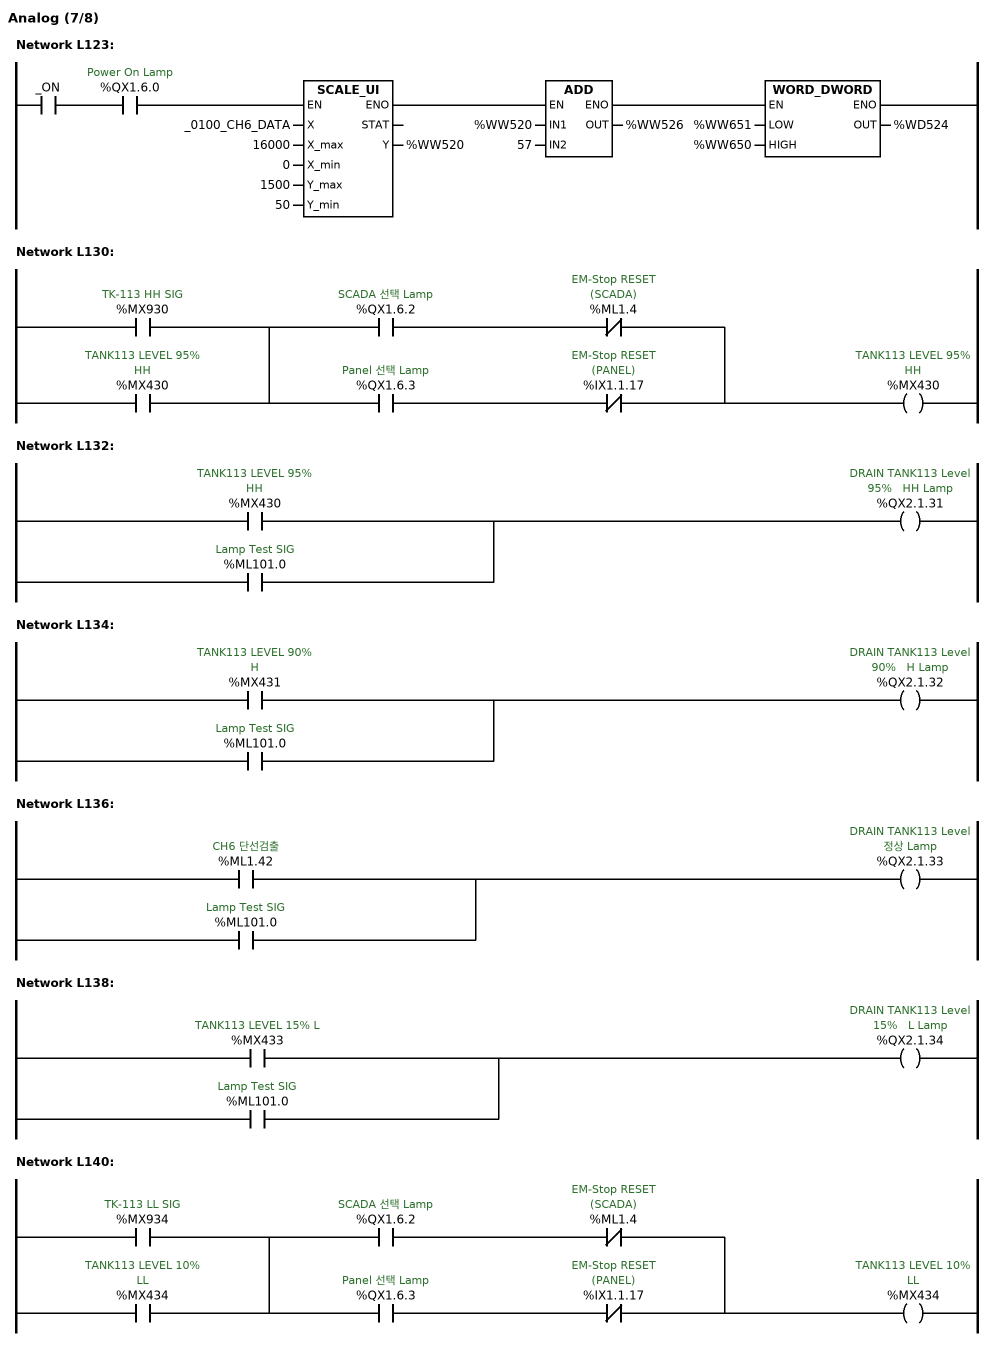
(* Rung L123 *)
IF _ON AND %QX1.6.0 THEN
    SCALE_UI(X := _0100_CH6_DATA, X_max := 16000, X_min := 0, Y_max := 1500, Y_min := 50, Y => %WW520);
    %WW526 := %WW520 + 57;
    %WD524 := WORD_DWORD(LOW := %WW651, HIGH := %WW650);
END_IF;
(* Rung L130 *)
%MX430 := (%MX930 OR %MX430) AND ((%QX1.6.2 AND NOT %ML1.4) OR (%QX1.6.3 AND NOT %IX1.1.17));
(* Rung L132 *)
%QX2.1.31 := %MX430 OR %ML101.0;
(* Rung L134 *)
%QX2.1.32 := %MX431 OR %ML101.0;
(* Rung L136 *)
%QX2.1.33 := %ML1.42 OR %ML101.0;
(* Rung L138 *)
%QX2.1.34 := %MX433 OR %ML101.0;
(* Rung L140 *)
%MX434 := (%MX934 OR %MX434) AND ((%QX1.6.2 AND NOT %ML1.4) OR (%QX1.6.3 AND NOT %IX1.1.17));

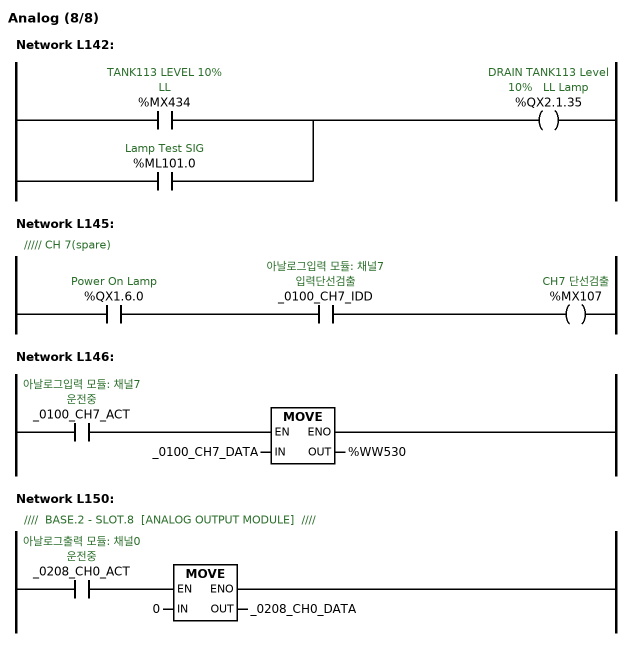
(* Rung L142 *)
%QX2.1.35 := %MX434 OR %ML101.0;
(* ///// CH 7(spare) *)
(* Rung L145 *)
%MX107 := %QX1.6.0 AND _0100_CH7_IDD;
(* Rung L146 *)
IF _0100_CH7_ACT THEN %WW530 := _0100_CH7_DATA; END_IF;
(* ////  BASE.2 - SLOT.8  [ANALOG OUTPUT MODULE]  //// *)
(* Rung L150 *)
IF _0208_CH0_ACT THEN _0208_CH0_DATA := 0; END_IF;
END_PROGRAM

PROGRAM Communication (* task: 스캔 프로그램 *)
(* PLC에서 컴퓨터로 데이타를 보냄 *)
VAR
    ATG_101 : TON;
    ATG_102 : TON;
    ATG_103 : TON;
    ATG_104 : TON;
    ATG_105 : TON;
    ATG_106 : TON;
    ATG_107 : TON;
    ATG_108 : TON;
    ATG_109 : TON;
    ATG_110 : TON;
    CM1 : TON;
    CM10 : TON;
    CM11 : TON;
    CM12 : TON;
    CM13 : TON;
    CM2 : TON;
    CM3 : TON;
    CM4 : TON;
    CM5 : TON;
    CM6 : TON;
    CM7 : TON;
    CM8 : TON;
    CM9 : TON;
    INST : TON;
    INST1 : TOF;
    P111A_FS : TON;
    P1O18A_FS : TON;
END_VAR
VAR_EXTERNAL
    _0000_ADDR_LNM : WORD; (* AT %LW3761 *) (* FEnet: LNM 정보(Ver 6.0이상) *)
    _0000_LINE_TOPOLOGY : BOOL; (* AT %LX60148 *) (* FEnet: Line topology 상태(Ver 6.0이상) *)
    _0100_CH0_ACT : BOOL; (* AT %UX1.0.16 *) (* 아날로그입력 모듈: 채널0 운전중 *)
    _0100_CH0_DATA : INT; (* AT %UW1.0.2 *) (* 아날로그입력 모듈: 채널0 변환값 *)
    _0100_CH1_DATA : INT; (* AT %UW1.0.3 *) (* 아날로그입력 모듈: 채널1 변환값 *)
    _0100_CH2_DATA : INT; (* AT %UW1.0.4 *) (* 아날로그입력 모듈: 채널2 변환값 *)
    _0100_CH3_DATA : INT; (* AT %UW1.0.5 *) (* 아날로그입력 모듈: 채널3 변환값 *)
    _0100_CH4_ACT : BOOL; (* AT %UX1.0.20 *) (* 아날로그입력 모듈: 채널4 운전중 *)
    _0100_CH4_DATA : INT; (* AT %UW1.0.6 *) (* 아날로그입력 모듈: 채널4 변환값 *)
    _0100_CH5_ACT : BOOL; (* AT %UX1.0.21 *) (* 아날로그입력 모듈: 채널5 운전중 *)
    _0100_CH5_DATA : INT; (* AT %UW1.0.7 *) (* 아날로그입력 모듈: 채널5 변환값 *)
    _0100_CH6_ACT : BOOL; (* AT %UX1.0.22 *) (* 아날로그입력 모듈: 채널6 운전중 *)
    _0100_CH6_DATA : INT; (* AT %UW1.0.8 *) (* 아날로그입력 모듈: 채널6 변환값 *)
END_VAR
VAR
    _t1 : BOOL;
    _t2 : BOOL;
    _t3 : BOOL;
    _t4 : BOOL;
    _t5 : BOOL;
    _t6 : BOOL;
    _t7 : BOOL;
    _t8 : BOOL;
    _t9 : BOOL;
    _t10 : BOOL;
END_VAR

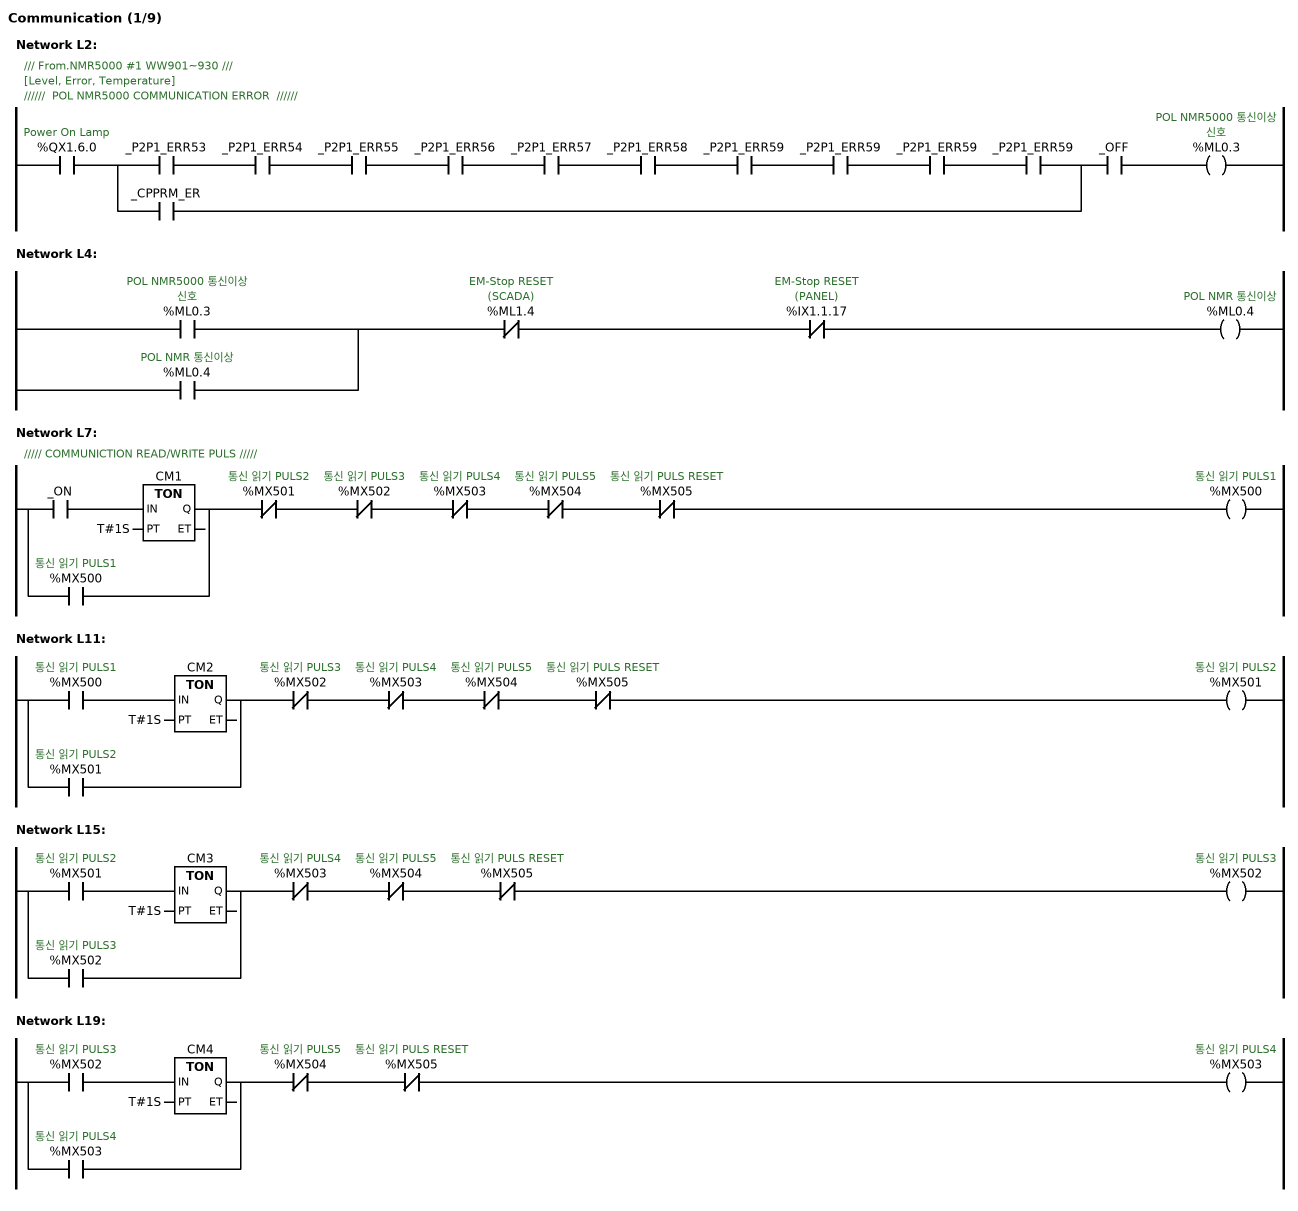
(* /// From.NMR5000 #1 WW901~930 /// / [Level, Error, Temperature] *)
(* //////  POL NMR5000 COMMUNICATION ERROR  ////// *)
(* Rung L2 *)
%ML0.3 := %QX1.6.0 AND ((_P2P1_ERR53 AND _P2P1_ERR54 AND _P2P1_ERR55 AND _P2P1_ERR56 AND _P2P1_ERR57 AND _P2P1_ERR58 AND _P2P1_ERR59 AND _P2P1_ERR59 AND _P2P1_ERR59 AND _P2P1_ERR59) OR _CPPRM_ER) AND _OFF;
(* Rung L4 *)
%ML0.4 := (%ML0.3 OR %ML0.4) AND NOT %ML1.4 AND NOT %IX1.1.17;
(* ///// COMMUNICTION READ/WRITE PULS ///// *)
(* Rung L7 *)
CM1(IN := _ON, PT := T#1S);
%MX500 := (CM1.Q OR %MX500) AND NOT %MX501 AND NOT %MX502 AND NOT %MX503 AND NOT %MX504 AND NOT %MX505;
(* Rung L11 *)
CM2(IN := %MX500, PT := T#1S);
%MX501 := (CM2.Q OR %MX501) AND NOT %MX502 AND NOT %MX503 AND NOT %MX504 AND NOT %MX505;
(* Rung L15 *)
CM3(IN := %MX501, PT := T#1S);
%MX502 := (CM3.Q OR %MX502) AND NOT %MX503 AND NOT %MX504 AND NOT %MX505;
(* Rung L19 *)
CM4(IN := %MX502, PT := T#1S);
%MX503 := (CM4.Q OR %MX503) AND NOT %MX504 AND NOT %MX505;

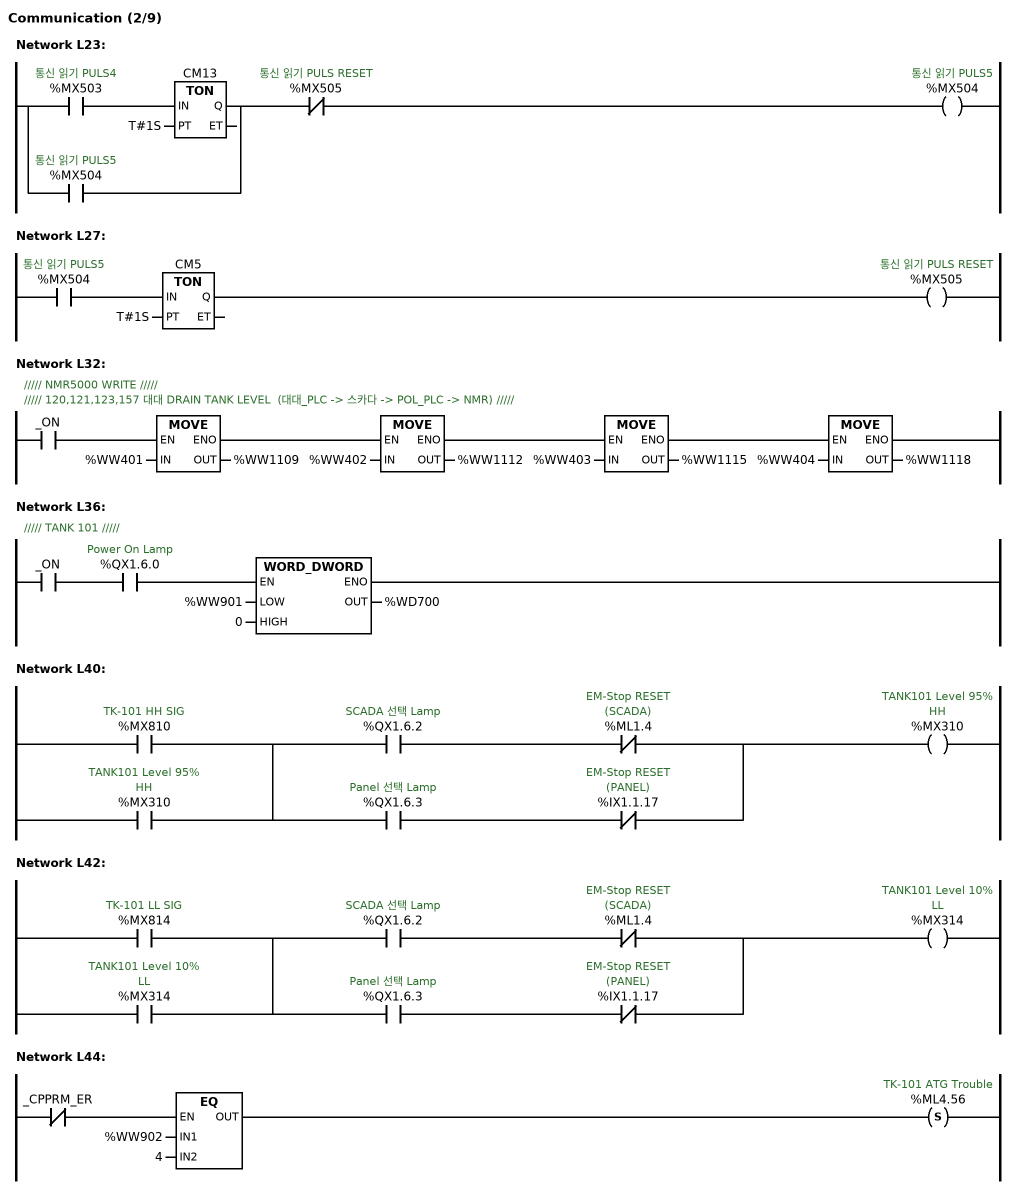
(* Rung L23 *)
CM13(IN := %MX503, PT := T#1S);
%MX504 := (CM13.Q OR %MX504) AND NOT %MX505;
(* Rung L27 *)
CM5(IN := %MX504, PT := T#1S);
%MX505 := CM5.Q;
(* ///// NMR5000 WRITE ///// *)
(* ///// 120,121,123,157 대대 DRAIN TANK LEVEL  (대대_PLC -> 스카다 -> POL_PLC -> NMR) ///// *)
(* Rung L32 *)
IF _ON THEN
    %WW1109 := %WW401;
    %WW1112 := %WW402;
    %WW1115 := %WW403;
    %WW1118 := %WW404;
END_IF;
(* ///// TANK 101 ///// *)
(* Rung L36 *)
IF _ON AND %QX1.6.0 THEN %WD700 := WORD_DWORD(LOW := %WW901, HIGH := 0); END_IF;
(* Rung L40 *)
%MX310 := (%MX810 OR %MX310) AND ((%QX1.6.2 AND NOT %ML1.4) OR (%QX1.6.3 AND NOT %IX1.1.17));
(* Rung L42 *)
%MX314 := (%MX814 OR %MX314) AND ((%QX1.6.2 AND NOT %ML1.4) OR (%QX1.6.3 AND NOT %IX1.1.17));
(* Rung L44 *)
IF NOT _CPPRM_ER THEN _t1 := %WW902 = 4; END_IF;
IF _t1 THEN %ML4.56 := TRUE; END_IF;

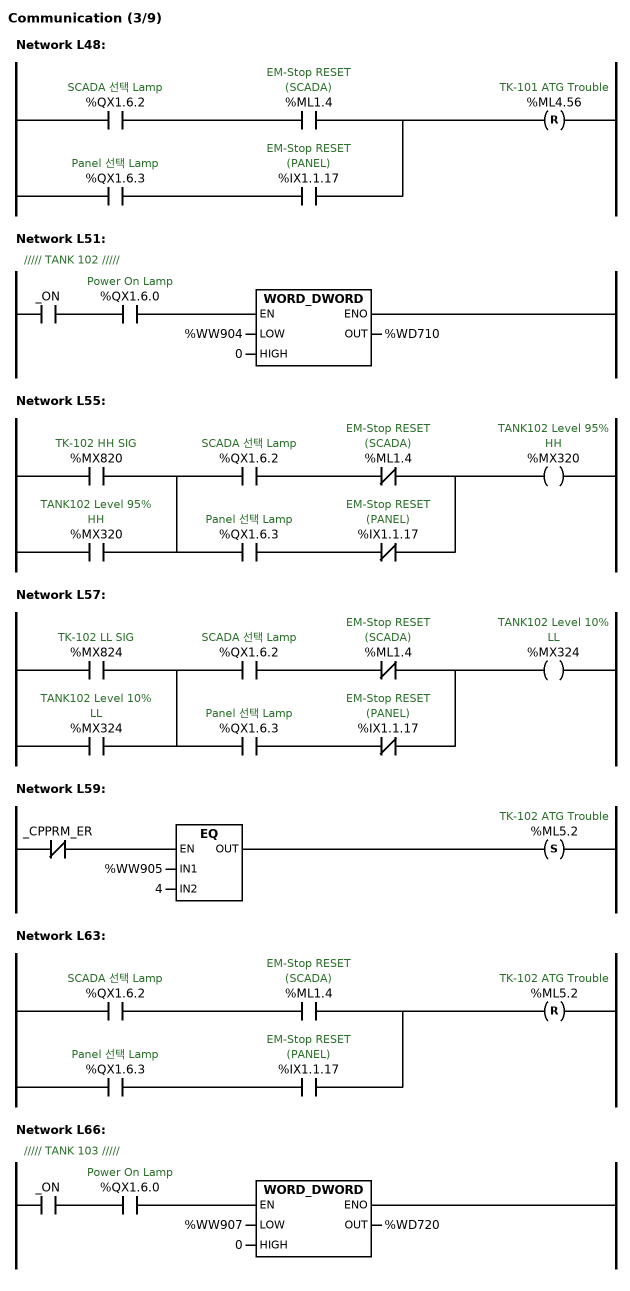
(* Rung L48 *)
IF (%QX1.6.2 AND %ML1.4) OR (%QX1.6.3 AND %IX1.1.17) THEN %ML4.56 := FALSE; END_IF;
(* ///// TANK 102 ///// *)
(* Rung L51 *)
IF _ON AND %QX1.6.0 THEN %WD710 := WORD_DWORD(LOW := %WW904, HIGH := 0); END_IF;
(* Rung L55 *)
%MX320 := (%MX820 OR %MX320) AND ((%QX1.6.2 AND NOT %ML1.4) OR (%QX1.6.3 AND NOT %IX1.1.17));
(* Rung L57 *)
%MX324 := (%MX824 OR %MX324) AND ((%QX1.6.2 AND NOT %ML1.4) OR (%QX1.6.3 AND NOT %IX1.1.17));
(* Rung L59 *)
IF NOT _CPPRM_ER THEN _t2 := %WW905 = 4; END_IF;
IF _t2 THEN %ML5.2 := TRUE; END_IF;
(* Rung L63 *)
IF (%QX1.6.2 AND %ML1.4) OR (%QX1.6.3 AND %IX1.1.17) THEN %ML5.2 := FALSE; END_IF;
(* ///// TANK 103 ///// *)
(* Rung L66 *)
IF _ON AND %QX1.6.0 THEN %WD720 := WORD_DWORD(LOW := %WW907, HIGH := 0); END_IF;

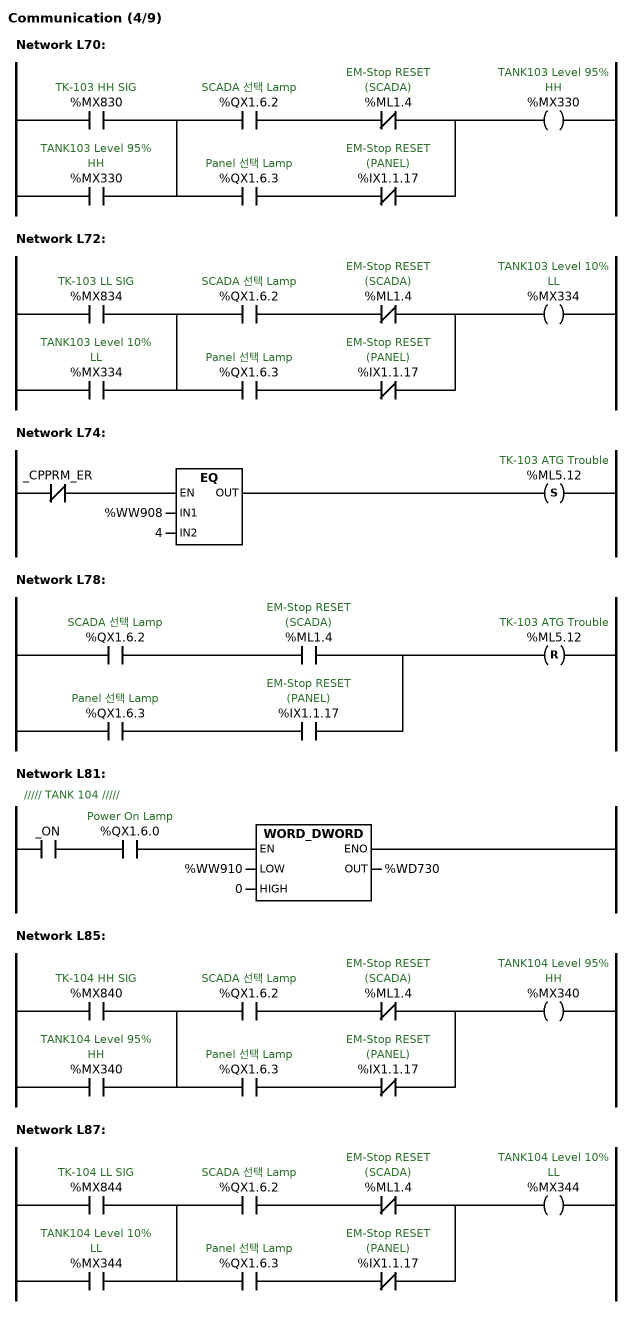
(* Rung L70 *)
%MX330 := (%MX830 OR %MX330) AND ((%QX1.6.2 AND NOT %ML1.4) OR (%QX1.6.3 AND NOT %IX1.1.17));
(* Rung L72 *)
%MX334 := (%MX834 OR %MX334) AND ((%QX1.6.2 AND NOT %ML1.4) OR (%QX1.6.3 AND NOT %IX1.1.17));
(* Rung L74 *)
IF NOT _CPPRM_ER THEN _t3 := %WW908 = 4; END_IF;
IF _t3 THEN %ML5.12 := TRUE; END_IF;
(* Rung L78 *)
IF (%QX1.6.2 AND %ML1.4) OR (%QX1.6.3 AND %IX1.1.17) THEN %ML5.12 := FALSE; END_IF;
(* ///// TANK 104 ///// *)
(* Rung L81 *)
IF _ON AND %QX1.6.0 THEN %WD730 := WORD_DWORD(LOW := %WW910, HIGH := 0); END_IF;
(* Rung L85 *)
%MX340 := (%MX840 OR %MX340) AND ((%QX1.6.2 AND NOT %ML1.4) OR (%QX1.6.3 AND NOT %IX1.1.17));
(* Rung L87 *)
%MX344 := (%MX844 OR %MX344) AND ((%QX1.6.2 AND NOT %ML1.4) OR (%QX1.6.3 AND NOT %IX1.1.17));

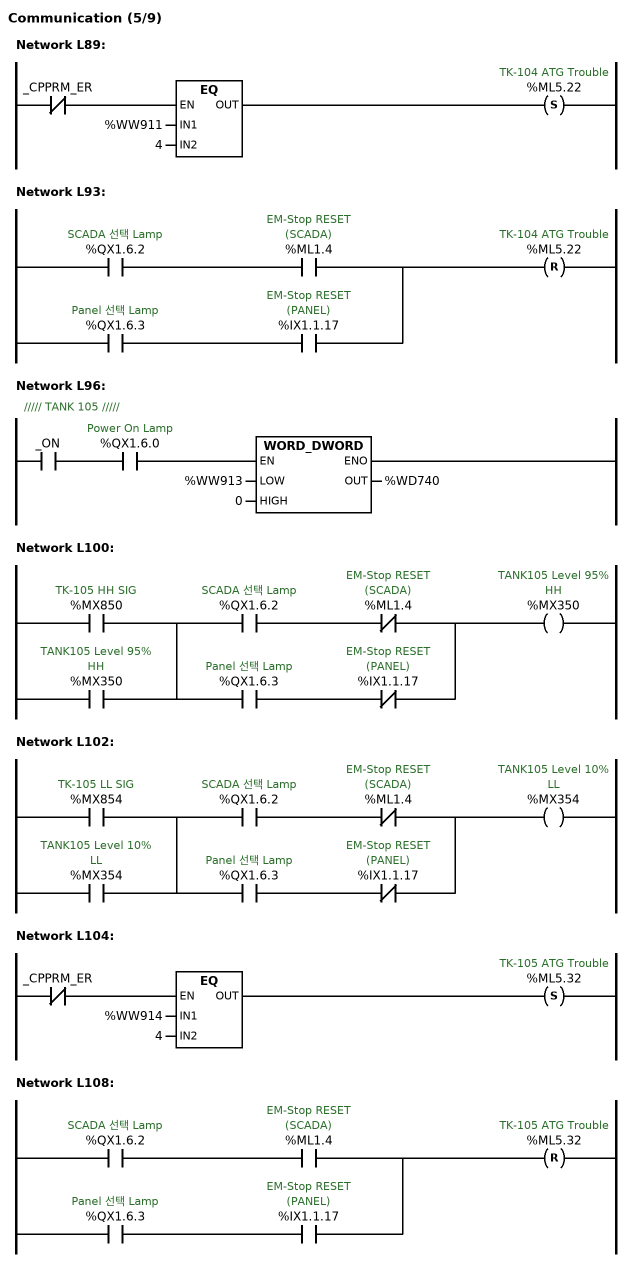
(* Rung L89 *)
IF NOT _CPPRM_ER THEN _t4 := %WW911 = 4; END_IF;
IF _t4 THEN %ML5.22 := TRUE; END_IF;
(* Rung L93 *)
IF (%QX1.6.2 AND %ML1.4) OR (%QX1.6.3 AND %IX1.1.17) THEN %ML5.22 := FALSE; END_IF;
(* ///// TANK 105 ///// *)
(* Rung L96 *)
IF _ON AND %QX1.6.0 THEN %WD740 := WORD_DWORD(LOW := %WW913, HIGH := 0); END_IF;
(* Rung L100 *)
%MX350 := (%MX850 OR %MX350) AND ((%QX1.6.2 AND NOT %ML1.4) OR (%QX1.6.3 AND NOT %IX1.1.17));
(* Rung L102 *)
%MX354 := (%MX854 OR %MX354) AND ((%QX1.6.2 AND NOT %ML1.4) OR (%QX1.6.3 AND NOT %IX1.1.17));
(* Rung L104 *)
IF NOT _CPPRM_ER THEN _t5 := %WW914 = 4; END_IF;
IF _t5 THEN %ML5.32 := TRUE; END_IF;
(* Rung L108 *)
IF (%QX1.6.2 AND %ML1.4) OR (%QX1.6.3 AND %IX1.1.17) THEN %ML5.32 := FALSE; END_IF;

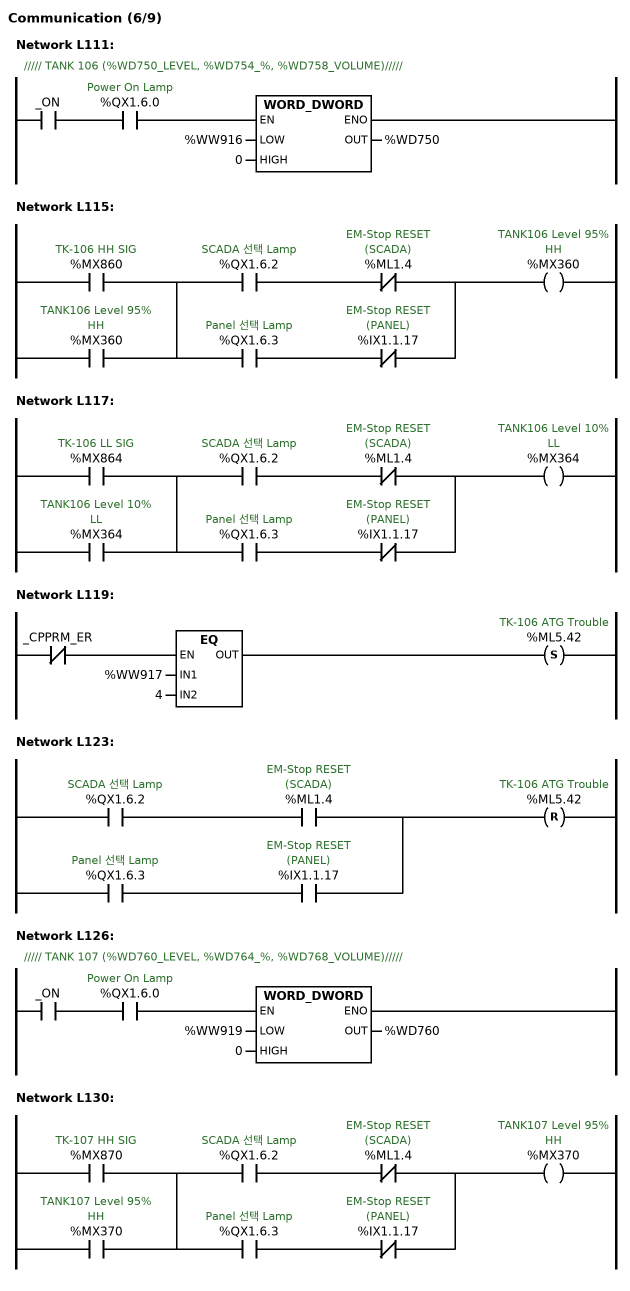
(* ///// TANK 106 (%WD750_LEVEL, %WD754_%, %WD758_VOLUME)///// *)
(* Rung L111 *)
IF _ON AND %QX1.6.0 THEN %WD750 := WORD_DWORD(LOW := %WW916, HIGH := 0); END_IF;
(* Rung L115 *)
%MX360 := (%MX860 OR %MX360) AND ((%QX1.6.2 AND NOT %ML1.4) OR (%QX1.6.3 AND NOT %IX1.1.17));
(* Rung L117 *)
%MX364 := (%MX864 OR %MX364) AND ((%QX1.6.2 AND NOT %ML1.4) OR (%QX1.6.3 AND NOT %IX1.1.17));
(* Rung L119 *)
IF NOT _CPPRM_ER THEN _t6 := %WW917 = 4; END_IF;
IF _t6 THEN %ML5.42 := TRUE; END_IF;
(* Rung L123 *)
IF (%QX1.6.2 AND %ML1.4) OR (%QX1.6.3 AND %IX1.1.17) THEN %ML5.42 := FALSE; END_IF;
(* ///// TANK 107 (%WD760_LEVEL, %WD764_%, %WD768_VOLUME)///// *)
(* Rung L126 *)
IF _ON AND %QX1.6.0 THEN %WD760 := WORD_DWORD(LOW := %WW919, HIGH := 0); END_IF;
(* Rung L130 *)
%MX370 := (%MX870 OR %MX370) AND ((%QX1.6.2 AND NOT %ML1.4) OR (%QX1.6.3 AND NOT %IX1.1.17));

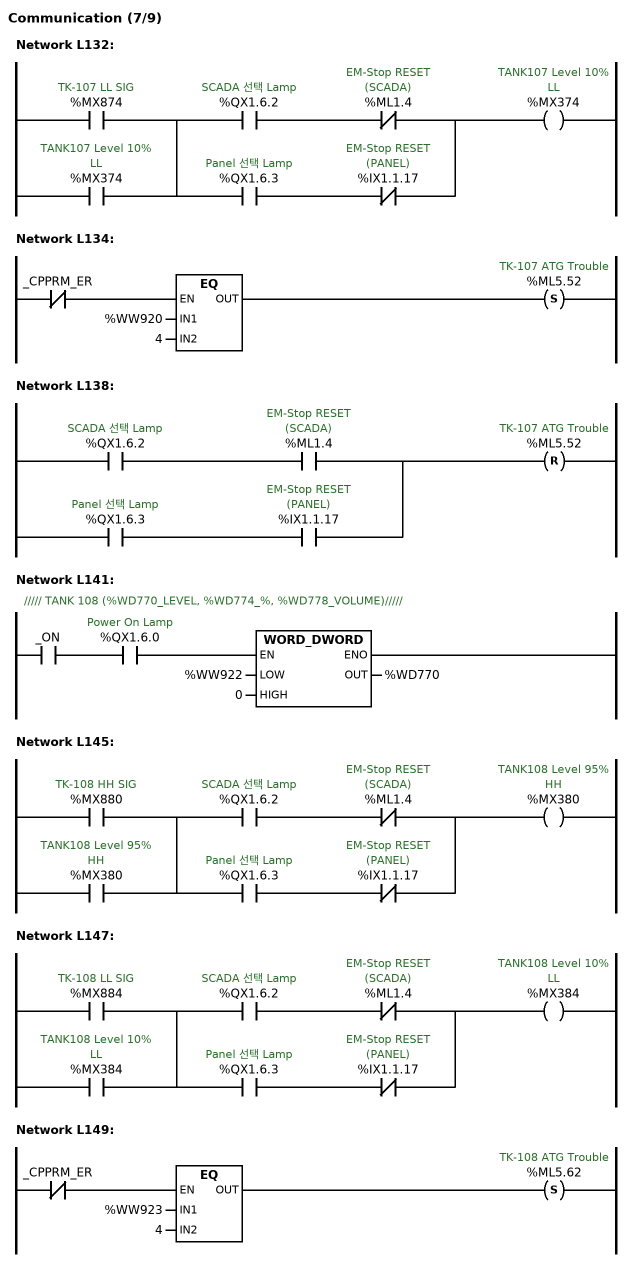
(* Rung L132 *)
%MX374 := (%MX874 OR %MX374) AND ((%QX1.6.2 AND NOT %ML1.4) OR (%QX1.6.3 AND NOT %IX1.1.17));
(* Rung L134 *)
IF NOT _CPPRM_ER THEN _t7 := %WW920 = 4; END_IF;
IF _t7 THEN %ML5.52 := TRUE; END_IF;
(* Rung L138 *)
IF (%QX1.6.2 AND %ML1.4) OR (%QX1.6.3 AND %IX1.1.17) THEN %ML5.52 := FALSE; END_IF;
(* ///// TANK 108 (%WD770_LEVEL, %WD774_%, %WD778_VOLUME)///// *)
(* Rung L141 *)
IF _ON AND %QX1.6.0 THEN %WD770 := WORD_DWORD(LOW := %WW922, HIGH := 0); END_IF;
(* Rung L145 *)
%MX380 := (%MX880 OR %MX380) AND ((%QX1.6.2 AND NOT %ML1.4) OR (%QX1.6.3 AND NOT %IX1.1.17));
(* Rung L147 *)
%MX384 := (%MX884 OR %MX384) AND ((%QX1.6.2 AND NOT %ML1.4) OR (%QX1.6.3 AND NOT %IX1.1.17));
(* Rung L149 *)
IF NOT _CPPRM_ER THEN _t8 := %WW923 = 4; END_IF;
IF _t8 THEN %ML5.62 := TRUE; END_IF;

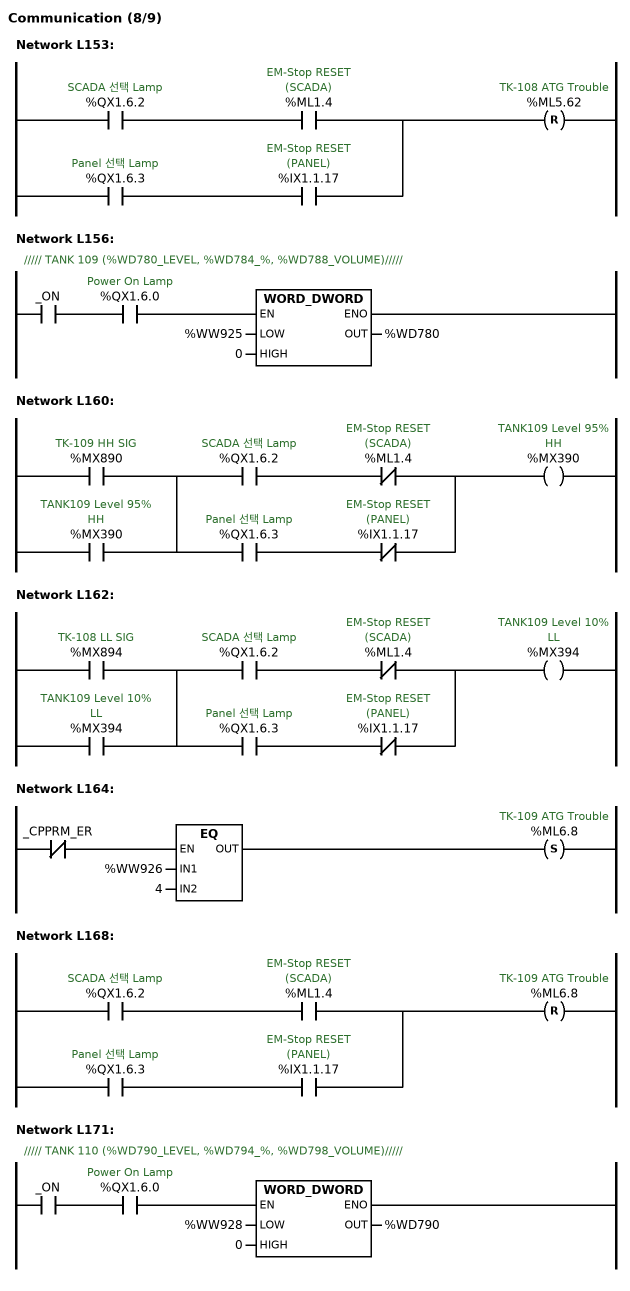
(* Rung L153 *)
IF (%QX1.6.2 AND %ML1.4) OR (%QX1.6.3 AND %IX1.1.17) THEN %ML5.62 := FALSE; END_IF;
(* ///// TANK 109 (%WD780_LEVEL, %WD784_%, %WD788_VOLUME)///// *)
(* Rung L156 *)
IF _ON AND %QX1.6.0 THEN %WD780 := WORD_DWORD(LOW := %WW925, HIGH := 0); END_IF;
(* Rung L160 *)
%MX390 := (%MX890 OR %MX390) AND ((%QX1.6.2 AND NOT %ML1.4) OR (%QX1.6.3 AND NOT %IX1.1.17));
(* Rung L162 *)
%MX394 := (%MX894 OR %MX394) AND ((%QX1.6.2 AND NOT %ML1.4) OR (%QX1.6.3 AND NOT %IX1.1.17));
(* Rung L164 *)
IF NOT _CPPRM_ER THEN _t9 := %WW926 = 4; END_IF;
IF _t9 THEN %ML6.8 := TRUE; END_IF;
(* Rung L168 *)
IF (%QX1.6.2 AND %ML1.4) OR (%QX1.6.3 AND %IX1.1.17) THEN %ML6.8 := FALSE; END_IF;
(* ///// TANK 110 (%WD790_LEVEL, %WD794_%, %WD798_VOLUME)///// *)
(* Rung L171 *)
IF _ON AND %QX1.6.0 THEN %WD790 := WORD_DWORD(LOW := %WW928, HIGH := 0); END_IF;

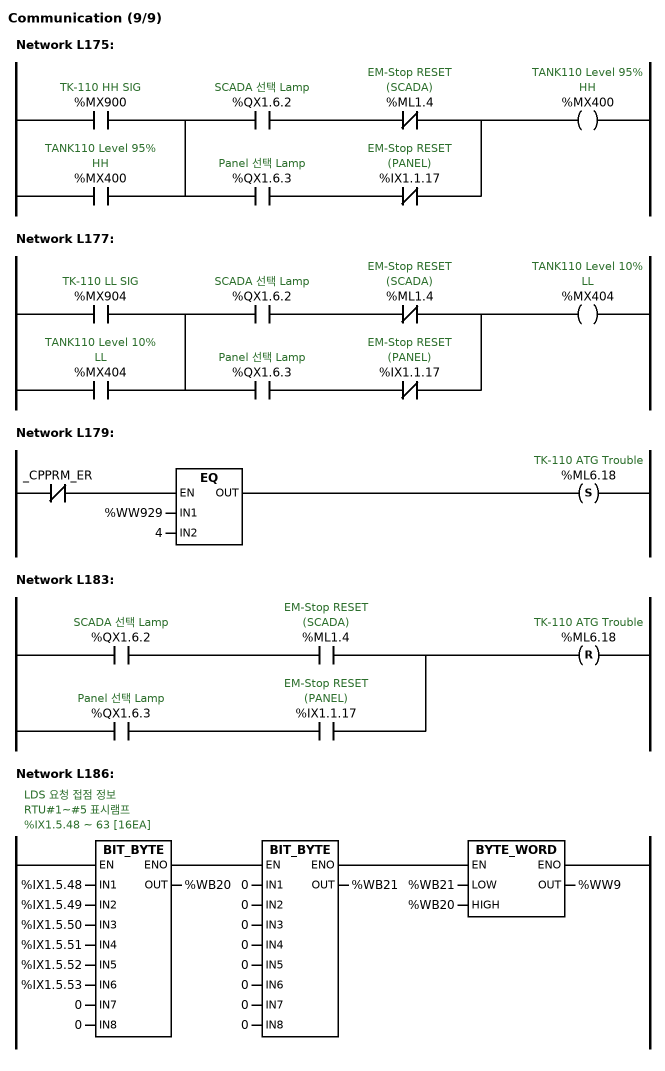
(* Rung L175 *)
%MX400 := (%MX900 OR %MX400) AND ((%QX1.6.2 AND NOT %ML1.4) OR (%QX1.6.3 AND NOT %IX1.1.17));
(* Rung L177 *)
%MX404 := (%MX904 OR %MX404) AND ((%QX1.6.2 AND NOT %ML1.4) OR (%QX1.6.3 AND NOT %IX1.1.17));
(* Rung L179 *)
IF NOT _CPPRM_ER THEN _t10 := %WW929 = 4; END_IF;
IF _t10 THEN %ML6.18 := TRUE; END_IF;
(* Rung L183 *)
IF (%QX1.6.2 AND %ML1.4) OR (%QX1.6.3 AND %IX1.1.17) THEN %ML6.18 := FALSE; END_IF;
(* LDS 요청 접점 정보 / RTU#1~#5 표시램프 / %IX1.5.48 ~ 63 [16EA] *)
(* Rung L186 *)
%WB20 := BIT_BYTE(%IX1.5.48, %IX1.5.49, %IX1.5.50, %IX1.5.51, %IX1.5.52, %IX1.5.53, 0, 0);
%WB21 := BIT_BYTE(0, 0, 0, 0, 0, 0, 0, 0);
%WW9 := BYTE_WORD(LOW := %WB21, HIGH := %WB20);
END_PROGRAM

PROGRAM Scada (* task: 스캔 프로그램 *)
VAR
    INST : TOF;
    INST1 : TOF;
    INST2 : TOF;
    INST3 : TOF;
    INST4 : TOF;
    INST5 : TOF;
END_VAR
VAR_EXTERNAL
    _0100_CH6_DATA : INT; (* AT %UW1.0.8 *) (* 아날로그입력 모듈: 채널6 변환값 *)
END_VAR

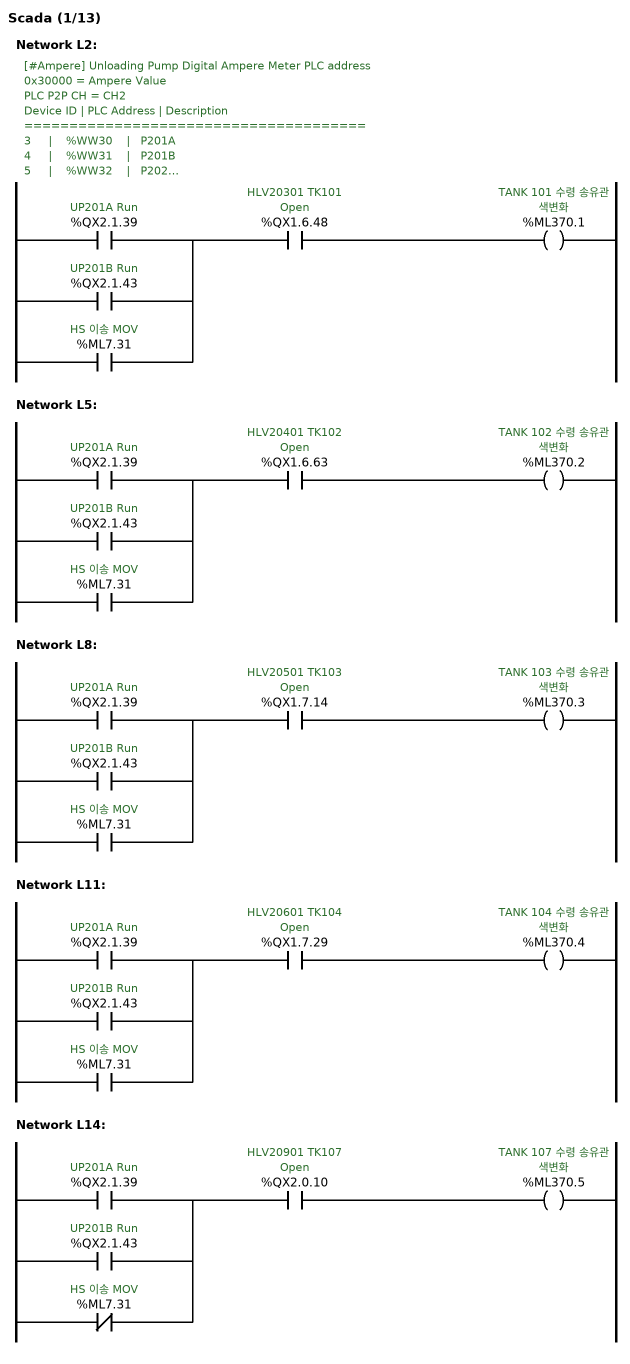
(* [#Ampere] Unloading Pump Digital Ampere Meter PLC address / 0x30000 = Ampere Value / PLC P2P CH = CH2 / Device ID | PLC Address | Description / ====================================== / 3     |    %WW30    |   P201A / 4     |    %WW31    |   P201B / 5     |    %WW32    |   P202A / 6     |    %WW33    |   P202B / 7     |    %WW34    |   P203A / 8     |    %WW35    |   P203B / ======================================= *)
(* **********   SCADA 송유관로 색변화     ********** *)
(* Rung L2 *)
%ML370.1 := (%QX2.1.39 OR %QX2.1.43 OR %ML7.31) AND %QX1.6.48;
(* Rung L5 *)
%ML370.2 := (%QX2.1.39 OR %QX2.1.43 OR %ML7.31) AND %QX1.6.63;
(* Rung L8 *)
%ML370.3 := (%QX2.1.39 OR %QX2.1.43 OR %ML7.31) AND %QX1.7.14;
(* Rung L11 *)
%ML370.4 := (%QX2.1.39 OR %QX2.1.43 OR %ML7.31) AND %QX1.7.29;
(* Rung L14 *)
%ML370.5 := (%QX2.1.39 OR %QX2.1.43 OR NOT %ML7.31) AND %QX2.0.10;

